LIN {X 0.001,Y -166.682,Z 591.348,A 0.000,B 0.000,C 90.000,E1 242.692} C_DIS
LIN {X -0.008,Y -162.664,Z 591.324,A 0.000,B 0.000,C 90.000,E1 238.329} C_DIS
LIN {X -0.035,Y -161.353,Z 591.314,A 0.000,B 0.000,C 90.000,E1 236.580} C_DIS
LIN {X -0.001,Y -157.347,Z 591.290,A 0.000,B 0.000,C 90.000,E1 232.145} C_DIS
LIN {X 0.028,Y -155.334,Z 591.275,A 0.000,B 0.000,C 90.000,E1 229.461} C_DIS
LIN {X -0.042,Y -151.684,Z 591.250,A 0.000,B 0.000,C 90.000,E1 225.000} C_DIS
LIN {X 0.006,Y -150.547,Z 591.240,A 0.000,B 0.000,C 90.000,E1 223.176} C_DIS
LIN {X 0.039,Y -147.274,Z 591.215,A 0.000,B 0.000,C 90.000,E1 218.624} C_DIS
LIN {X 0.012,Y -145.301,Z 591.194,A 0.000,B 0.000,C 90.000,E1 214.978} C_DIS
LIN {X 0.004,Y -142.395,Z 591.164,A 0.000,B 0.000,C 90.000,E1 209.461} C_DIS
LIN {X -0.014,Y -141.376,Z 591.148,A 0.000,B 0.000,C 90.000,E1 206.693} C_DIS
LIN {X 0.028,Y -139.348,Z 591.112,A 0.000,B 0.000,C 90.000,E1 200.174} C_DIS
LIN {X -0.031,Y -138.784,Z 591.097,A 0.000,B 0.000,C 90.000,E1 197.402} C_DIS
LIN {X 0.028,Y -138.343,Z 591.055,A 0.000,B 0.000,C 90.000,E1 189.905} C_DIS
LIN {X 0.048,Y -139.390,Z 591.008,A 0.000,B 0.000,C 90.000,E1 181.489} C_DIS
LIN {X -0.039,Y -141.288,Z 590.972,A 0.000,B 0.000,C 90.000,E1 175.008} C_DIS
LIN {X 0.061,Y -142.651,Z 590.957,A 0.000,B 0.000,C 90.000,E1 172.186} C_DIS
LIN {X 0.010,Y -144.990,Z 590.931,A 0.000,B 0.000,C 90.000,E1 167.589} C_DIS
LIN {X 0.001,Y -147.617,Z 590.911,A 0.000,B 0.000,C 90.000,E1 163.921} C_DIS
LIN {X 0.079,Y -150.242,Z 590.890,A 0.000,B 0.000,C 90.000,E1 160.242} C_DIS
LIN {X -0.047,Y -153.635,Z 590.870,A 0.000,B 0.000,C 90.000,E1 156.666} C_DIS
LIN {X 0.011,Y -157.051,Z 590.850,A 0.000,B 0.000,C 90.000,E1 153.050} C_DIS
LIN {X 0.009,Y -161.179,Z 590.831,A 0.000,B 0.000,C 90.000,E1 149.488} C_DIS
LIN {X 0.039,Y -163.273,Z 590.821,A 0.000,B 0.000,C 90.000,E1 147.709} C_DIS
LIN {X 0.050,Y -167.715,Z 590.801,A 0.000,B 0.000,C 90.000,E1 144.196} C_DIS
LIN {X -0.037,Y -171.534,Z 590.787,A 0.000,B 0.000,C 90.000,E1 141.618} C_DIS
LIN {X 0.006,Y -176.474,Z 590.768,A 0.000,B 0.000,C 90.000,E1 138.162} C_DIS
LIN {X 0.005,Y -180.771,Z 590.753,A 0.000,B 0.000,C 90.000,E1 135.607} C_DIS
LIN {X -0.008,Y -186.178,Z 590.735,A 0.000,B 0.000,C 90.000,E1 132.243} C_DIS
LIN {X -0.017,Y -191.384,Z 590.719,A 0.000,B 0.000,C 90.000,E1 129.402} C_DIS
LIN {X -0.061,Y -288.933,Z 590.719,A 0.000,B 0.000,C 90.000,E1 129.402} C_DIS
LIN {X -0.121,Y -291.320,Z 590.719,A 0.000,B 0.000,C 90.000,E1 129.358} C_DIS
LIN {X 0.044,Y -295.133,Z 590.717,A 0.000,B 0.000,C 90.000,E1 129.116} C_DIS
LIN {X 0.024,Y -297.460,Z 590.716,A 0.000,B 0.000,C 90.000,E1 128.910} C_DIS
LIN {X 0.053,Y -301.291,Z 590.713,A 0.000,B 0.000,C 90.000,E1 128.382} C_DIS
LIN {X 0.049,Y -302.982,Z 590.711,A 0.000,B 0.000,C 90.000,E1 128.051} C_DIS
LIN {X -0.008,Y -304.309,Z 590.710,A 0.000,B 0.000,C 90.000,E1 127.729} C_DIS
LIN {X 0.022,Y -313.953,Z 590.691,A 0.000,B 0.000,C 90.000,E1 124.452} C_DIS
LIN {X 0.123,Y -323.776,Z 590.675,A 0.000,B 0.000,C 90.000,E1 121.544} C_DIS
LIN {X -0.106,Y -334.914,Z 590.660,A 0.000,B 0.000,C 90.000,E1 118.743} C_DIS
LIN {X 0.095,Y -347.463,Z 590.644,A 0.000,B 0.000,C 90.000,E1 115.924} C_DIS
LIN {X -0.003,Y -359.895,Z 590.631,A 0.000,B 0.000,C 90.000,E1 113.515} C_DIS
LIN {X -0.093,Y -373.621,Z 590.617,A 0.000,B 0.000,C 90.000,E1 111.153} C_DIS
LIN {X -0.121,Y -388.742,Z 590.605,A 0.000,B 0.000,C 90.000,E1 108.833} C_DIS
LIN {X -0.019,Y -405.367,Z 590.592,A 0.000,B 0.000,C 90.000,E1 106.551} C_DIS
LIN {X -0.121,Y -423.616,Z 590.580,A 0.000,B 0.000,C 90.000,E1 104.356} C_DIS
LIN {X -0.201,Y -443.370,Z 590.568,A 0.000,B 0.000,C 90.000,E1 102.243} C_DIS
LIN {X 0.076,Y -463.790,Z 590.557,A 0.000,B 0.000,C 90.000,E1 100.254} C_DIS
LIN {X 0.219,Y -474.052,Z 590.552,A 0.000,B 0.000,C 90.000,E1 99.321} C_DIS
LIN {X -0.232,Y -475.936,Z 590.551,A 0.000,B 0.000,C 90.000,E1 99.151} C_DIS
LIN {X 0.102,Y -477.544,Z 590.549,A 0.000,B 0.000,C 90.000,E1 98.859} C_DIS
LIN {X -0.036,Y -478.750,Z 590.548,A 0.000,B 0.000,C 90.000,E1 98.624} C_DIS
LIN {X 0.110,Y -480.218,Z 590.545,A 0.000,B 0.000,C 90.000,E1 98.106} C_DIS
LIN {X -0.212,Y -480.647,Z 590.542,A 0.000,B 0.000,C 90.000,E1 97.644} C_DIS
LIN {X -0.048,Y -480.105,Z 590.540,A 0.000,B 0.000,C 90.000,E1 97.125} C_DIS
LIN {X 0.119,Y -478.511,Z 590.537,A 0.000,B 0.000,C 90.000,E1 96.606} C_DIS
LIN {X -0.010,Y -477.230,Z 590.535,A 0.000,B 0.000,C 90.000,E1 96.372} C_DIS
LIN {X 0.142,Y -473.633,Z 590.533,A 0.000,B 0.000,C 90.000,E1 95.853} C_DIS
LIN {X 0.030,Y -459.012,Z 590.521,A 0.000,B 0.000,C 90.000,E1 93.841} C_DIS
LIN {X -0.195,Y -447.691,Z 590.511,A 0.000,B 0.000,C 90.000,E1 92.064} C_DIS
LIN {X -0.018,Y -436.085,Z 590.500,A 0.000,B 0.000,C 90.000,E1 89.943} C_DIS
LIN {X -0.110,Y -428.555,Z 590.492,A 0.000,B 0.000,C 90.000,E1 88.625} C_DIS
LIN {X -0.182,Y -419.081,Z 590.483,A 0.000,B 0.000,C 90.000,E1 87.020} C_DIS
LIN {X -0.058,Y -403.319,Z 590.468,A 0.000,B 0.000,C 90.000,E1 84.261} C_DIS
LIN {X 0.032,Y -389.890,Z 590.454,A 0.000,B 0.000,C 90.000,E1 81.724} C_DIS
LIN {X -0.088,Y -378.203,Z 590.441,A 0.000,B 0.000,C 90.000,E1 79.454} C_DIS
LIN {X -0.056,Y -365.412,Z 590.427,A 0.000,B 0.000,C 90.000,E1 76.825} C_DIS
LIN {X -0.079,Y -351.916,Z 590.410,A 0.000,B 0.000,C 90.000,E1 73.850} C_DIS
LIN {X 0.043,Y -339.732,Z 590.393,A 0.000,B 0.000,C 90.000,E1 70.786} C_DIS
LIN {X 0.158,Y -329.793,Z 590.378,A 0.000,B 0.000,C 90.000,E1 67.975} C_DIS
LIN {X 0.040,Y -319.831,Z 590.360,A 0.000,B 0.000,C 90.000,E1 64.845} C_DIS
LIN {X 0.058,Y -312.250,Z 590.346,A 0.000,B 0.000,C 90.000,E1 62.281} C_DIS
LIN {X 0.176,Y -304.903,Z 590.332,A 0.000,B 0.000,C 90.000,E1 59.665} C_DIS
LIN {X 0.152,Y -297.769,Z 590.317,A 0.000,B 0.000,C 90.000,E1 57.041} C_DIS
LIN {X -0.058,Y -289.305,Z 590.299,A 0.000,B 0.000,C 90.000,E1 53.749} C_DIS
LIN {X 0.077,Y -284.390,Z 590.287,A 0.000,B 0.000,C 90.000,E1 51.698} C_DIS
LIN {X 0.022,Y -279.299,Z 590.276,A 0.000,B 0.000,C 90.000,E1 49.666} C_DIS
LIN {X -0.123,Y -275.670,Z 590.268,A 0.000,B 0.000,C 90.000,E1 48.324} C_DIS
LIN {X 0.052,Y -271.817,Z 590.261,A 0.000,B 0.000,C 90.000,E1 46.905} C_DIS
LIN {X -0.010,Y -267.604,Z 590.253,A 0.000,B 0.000,C 90.000,E1 45.526} C_DIS
LIN {X -0.022,Y -260.833,Z 590.241,A 0.000,B 0.000,C 90.000,E1 43.419} C_DIS
LIN {X 0.032,Y -252.799,Z 590.227,A 0.000,B 0.000,C 90.000,E1 40.906} C_DIS
LIN {X -0.030,Y -242.966,Z 590.209,A 0.000,B 0.000,C 90.000,E1 37.649} C_DIS
LIN {X -0.027,Y -235.024,Z 590.193,A 0.000,B 0.000,C 90.000,E1 34.692} C_DIS
LIN {X 0.037,Y -227.788,Z 590.176,A 0.000,B 0.000,C 90.000,E1 31.671} C_DIS
LIN {X 0.065,Y -221.233,Z 590.159,A 0.000,B 0.000,C 90.000,E1 28.615} C_DIS
LIN {X 0.005,Y -215.441,Z 590.142,A 0.000,B 0.000,C 90.000,E1 25.540} C_DIS
LIN {X 0.018,Y -210.399,Z 590.125,A 0.000,B 0.000,C 90.000,E1 22.408} C_DIS
LIN {X -0.052,Y -205.263,Z 590.103,A 0.000,B 0.000,C 90.000,E1 18.471} C_DIS
LIN {X -0.080,Y -201.272,Z 590.080,A 0.000,B 0.000,C 90.000,E1 14.481} C_DIS
LIN {X 0.013,Y -197.803,Z 590.053,A 0.000,B 0.000,C 90.000,E1 9.613} C_DIS
LIN {X 0.016,Y -195.578,Z 590.013,A 0.000,B 0.000,C 90.000,E1 2.293} C_DIS
LIN {X 0.101,Y -197.278,Z 589.966,A 0.000,B 0.000,C 90.000,E1 353.799} C_DIS
LIN {X -0.074,Y -200.204,Z 589.939,A 0.000,B 0.000,C 90.000,E1 348.982} C_DIS
LIN {X -0.099,Y -204.480,Z 589.912,A 0.000,B 0.000,C 90.000,E1 344.157} C_DIS
LIN {X 0.015,Y -208.872,Z 589.890,A 0.000,B 0.000,C 90.000,E1 340.134} C_DIS
LIN {X 0.037,Y -214.099,Z 589.868,A 0.000,B 0.000,C 90.000,E1 336.177} C_DIS
LIN {X -0.003,Y -220.025,Z 589.846,A 0.000,B 0.000,C 90.000,E1 332.281} C_DIS
LIN {X 0.066,Y -226.572,Z 589.825,A 0.000,B 0.000,C 90.000,E1 328.408} C_DIS
LIN {X -0.044,Y -232.201,Z 589.808,A 0.000,B 0.000,C 90.000,E1 325.388} C_DIS
LIN {X 0.004,Y -239.520,Z 589.787,A 0.000,B 0.000,C 90.000,E1 321.618} C_DIS
LIN {X -0.014,Y -247.551,Z 589.766,A 0.000,B 0.000,C 90.000,E1 317.919} C_DIS
LIN {X 0.014,Y -256.490,Z 589.746,A 0.000,B 0.000,C 90.000,E1 314.271} C_DIS
LIN {X -0.004,Y -266.682,Z 589.726,A 0.000,B 0.000,C 90.000,E1 310.701} C_DIS
LIN {X 0.028,Y -276.166,Z 589.711,A 0.000,B 0.000,C 90.000,E1 307.890} C_DIS
LIN {X -0.108,Y -289.433,Z 589.691,A 0.000,B 0.000,C 90.000,E1 304.485} C_DIS
LIN {X -0.071,Y -304.313,Z 589.673,A 0.000,B 0.000,C 90.000,E1 301.131} C_DIS
LIN {X 0.103,Y -317.089,Z 589.658,A 0.000,B 0.000,C 90.000,E1 298.487} C_DIS
LIN {X -0.070,Y -333.996,Z 589.641,A 0.000,B 0.000,C 90.000,E1 295.335} C_DIS
LIN {X 0.135,Y -348.856,Z 589.627,A 0.000,B 0.000,C 90.000,E1 292.823} C_DIS
LIN {X -0.003,Y -365.106,Z 589.613,A 0.000,B 0.000,C 90.000,E1 290.429} C_DIS
LIN {X 0.155,Y -385.211,Z 589.599,A 0.000,B 0.000,C 90.000,E1 287.764} C_DIS
LIN {X -0.042,Y -399.377,Z 589.589,A 0.000,B 0.000,C 90.000,E1 286.079} C_DIS
LIN {X -0.112,Y -413.409,Z 589.580,A 0.000,B 0.000,C 90.000,E1 284.411} C_DIS
LIN {X -0.131,Y -427.361,Z 589.571,A 0.000,B 0.000,C 90.000,E1 282.771} C_DIS
LIN {X 0.145,Y -436.179,Z 589.565,A 0.000,B 0.000,C 90.000,E1 281.658} C_DIS
LIN {X 0.101,Y -444.479,Z 589.559,A 0.000,B 0.000,C 90.000,E1 280.602} C_DIS
LIN {X 0.070,Y -452.385,Z 589.553,A 0.000,B 0.000,C 90.000,E1 279.557} C_DIS
LIN {X -0.139,Y -457.960,Z 589.549,A 0.000,B 0.000,C 90.000,E1 278.803} C_DIS
LIN {X -0.015,Y -464.839,Z 589.543,A 0.000,B 0.000,C 90.000,E1 277.757} C_DIS
LIN {X 0.129,Y -471.173,Z 589.537,A 0.000,B 0.000,C 90.000,E1 276.720} C_DIS
LIN {X 0.081,Y -475.463,Z 589.533,A 0.000,B 0.000,C 90.000,E1 275.967} C_DIS
LIN {X 0.013,Y -479.078,Z 589.529,A 0.000,B 0.000,C 90.000,E1 275.220} C_DIS
LIN {X 0.162,Y -481.108,Z 589.526,A 0.000,B 0.000,C 90.000,E1 274.702} C_DIS
LIN {X -0.200,Y -482.801,Z 589.523,A 0.000,B 0.000,C 90.000,E1 274.245} C_DIS
LIN {X -0.034,Y -484.173,Z 589.521,A 0.000,B 0.000,C 90.000,E1 273.726} C_DIS
LIN {X 0.112,Y -485.263,Z 589.518,A 0.000,B 0.000,C 90.000,E1 273.212} C_DIS
LIN {X -0.192,Y -486.019,Z 589.515,A 0.000,B 0.000,C 90.000,E1 272.751} C_DIS
LIN {X -0.028,Y -486.481,Z 589.512,A 0.000,B 0.000,C 90.000,E1 272.236} C_DIS
LIN {X 0.158,Y -486.570,Z 589.510,A 0.000,B 0.000,C 90.000,E1 271.718} C_DIS
LIN {X -0.157,Y -486.200,Z 589.507,A 0.000,B 0.000,C 90.000,E1 271.260} C_DIS
LIN {X 0.017,Y -485.368,Z 589.504,A 0.000,B 0.000,C 90.000,E1 270.745} C_DIS
LIN {X 0.189,Y -484.045,Z 589.501,A 0.000,B 0.000,C 90.000,E1 270.229} C_DIS
LIN {X -0.127,Y -482.086,Z 589.499,A 0.000,B 0.000,C 90.000,E1 269.771} C_DIS
LIN {X 0.032,Y -479.359,Z 589.496,A 0.000,B 0.000,C 90.000,E1 269.255} C_DIS
LIN {X -0.137,Y -477.707,Z 589.495,A 0.000,B 0.000,C 90.000,E1 269.026} C_DIS
LIN {X -0.008,Y -473.588,Z 589.492,A 0.000,B 0.000,C 90.000,E1 268.511} C_DIS
LIN {X -0.185,Y -471.206,Z 589.490,A 0.000,B 0.000,C 90.000,E1 268.282} C_DIS
LIN {X -0.073,Y -465.267,Z 589.488,A 0.000,B 0.000,C 90.000,E1 267.764} C_DIS
LIN {X 0.141,Y -458.882,Z 589.485,A 0.000,B 0.000,C 90.000,E1 267.306} C_DIS
LIN {X -0.018,Y -451.775,Z 589.483,A 0.000,B 0.000,C 90.000,E1 266.963} C_DIS
LIN {X 0.003,Y -444.612,Z 589.482,A 0.000,B 0.000,C 90.000,E1 266.674} C_DIS
LIN {X -0.015,Y -436.746,Z 589.480,A 0.000,B 0.000,C 90.000,E1 266.445} C_DIS
LIN {X -0.018,Y -428.223,Z 589.479,A 0.000,B 0.000,C 90.000,E1 266.274} C_DIS
LIN {X -0.045,Y -418.357,Z 589.479,A 0.000,B 0.000,C 90.000,E1 266.159} C_DIS
LIN {X -0.061,Y -408.534,Z 589.478,A 0.000,B 0.000,C 90.000,E1 266.102} C_DIS
LIN {X -0.058,Y -180.923,Z 589.478,A 0.000,B 0.000,C 90.000,E1 266.102} C_DIS
LIN {X -0.013,Y -180.875,Z 589.473,A 0.000,B 0.000,C 90.000,E1 265.065} C_DIS
LIN {X 0.069,Y -178.940,Z 589.443,A 0.000,B 0.000,C 90.000,E1 259.803} C_DIS
LIN {X -0.063,Y -175.990,Z 589.415,A 0.000,B 0.000,C 90.000,E1 254.755} C_DIS
LIN {X 0.052,Y -175.491,Z 589.410,A 0.000,B 0.000,C 90.000,E1 253.866} C_DIS
LIN {X -0.054,Y -172.235,Z 589.387,A 0.000,B 0.000,C 90.000,E1 249.625} C_DIS
LIN {X -0.075,Y -171.712,Z 589.382,A 0.000,B 0.000,C 90.000,E1 248.773} C_DIS
LIN {X 0.010,Y -167.307,Z 589.353,A 0.000,B 0.000,C 90.000,E1 243.563} C_DIS
LIN {X 0.016,Y -166.687,Z 589.348,A 0.000,B 0.000,C 90.000,E1 242.692} C_DIS
LIN {X 0.006,Y -162.668,Z 589.324,A 0.000,B 0.000,C 90.000,E1 238.329} C_DIS
LIN {X -0.020,Y -161.358,Z 589.314,A 0.000,B 0.000,C 90.000,E1 236.580} C_DIS
LIN {X 0.014,Y -157.351,Z 589.290,A 0.000,B 0.000,C 90.000,E1 232.145} C_DIS
LIN {X 0.043,Y -155.339,Z 589.275,A 0.000,B 0.000,C 90.000,E1 229.461} C_DIS
LIN {X -0.028,Y -151.688,Z 589.250,A 0.000,B 0.000,C 90.000,E1 225.000} C_DIS
LIN {X 0.021,Y -150.551,Z 589.240,A 0.000,B 0.000,C 90.000,E1 223.176} C_DIS
LIN {X 0.053,Y -147.277,Z 589.215,A 0.000,B 0.000,C 90.000,E1 218.624} C_DIS
LIN {X 0.026,Y -145.305,Z 589.194,A 0.000,B 0.000,C 90.000,E1 214.978} C_DIS
LIN {X 0.017,Y -142.398,Z 589.164,A 0.000,B 0.000,C 90.000,E1 209.461} C_DIS
LIN {X 0.000,Y -141.378,Z 589.148,A 0.000,B 0.000,C 90.000,E1 206.693} C_DIS
LIN {X 0.041,Y -139.348,Z 589.112,A 0.000,B 0.000,C 90.000,E1 200.174} C_DIS
LIN {X -0.018,Y -138.785,Z 589.097,A 0.000,B 0.000,C 90.000,E1 197.402} C_DIS
LIN {X 0.041,Y -138.344,Z 589.055,A 0.000,B 0.000,C 90.000,E1 189.905} C_DIS
LIN {X 0.062,Y -139.389,Z 589.008,A 0.000,B 0.000,C 90.000,E1 181.489} C_DIS
LIN {X -0.025,Y -141.285,Z 588.972,A 0.000,B 0.000,C 90.000,E1 175.008} C_DIS
LIN {X -0.067,Y -142.649,Z 588.957,A 0.000,B 0.000,C 90.000,E1 172.243} C_DIS
LIN {X 0.025,Y -144.986,Z 588.931,A 0.000,B 0.000,C 90.000,E1 167.589} C_DIS
LIN {X 0.014,Y -147.614,Z 588.911,A 0.000,B 0.000,C 90.000,E1 163.921} C_DIS
LIN {X -0.048,Y -150.237,Z 588.890,A 0.000,B 0.000,C 90.000,E1 160.296} C_DIS
LIN {X -0.032,Y -153.630,Z 588.870,A 0.000,B 0.000,C 90.000,E1 156.666} C_DIS
LIN {X 0.026,Y -157.046,Z 588.850,A 0.000,B 0.000,C 90.000,E1 153.050} C_DIS
LIN {X 0.025,Y -161.172,Z 588.831,A 0.000,B 0.000,C 90.000,E1 149.488} C_DIS
LIN {X -0.033,Y -163.267,Z 588.821,A 0.000,B 0.000,C 90.000,E1 147.740} C_DIS
LIN {X 0.066,Y -167.707,Z 588.801,A 0.000,B 0.000,C 90.000,E1 144.196} C_DIS
LIN {X -0.021,Y -171.527,Z 588.787,A 0.000,B 0.000,C 90.000,E1 141.618} C_DIS
LIN {X 0.022,Y -176.467,Z 588.768,A 0.000,B 0.000,C 90.000,E1 138.162} C_DIS
LIN {X -0.109,Y -180.763,Z 588.753,A 0.000,B 0.000,C 90.000,E1 135.648} C_DIS
LIN {X 0.010,Y -186.169,Z 588.735,A 0.000,B 0.000,C 90.000,E1 132.243} C_DIS
LIN {X -0.002,Y -191.377,Z 588.719,A 0.000,B 0.000,C 90.000,E1 129.402} C_DIS
LIN {X -0.048,Y -191.400,Z 588.719,A 0.000,B 0.000,C 90.000,E1 129.402} C_DIS
LIN {X 0.115,Y -288.729,Z 588.719,A 0.000,B 0.000,C 90.000,E1 129.358} C_DIS
LIN {X -0.096,Y -290.833,Z 588.719,A 0.000,B 0.000,C 90.000,E1 129.358} C_DIS
LIN {X 0.069,Y -294.924,Z 588.717,A 0.000,B 0.000,C 90.000,E1 129.116} C_DIS
LIN {X 0.050,Y -297.311,Z 588.716,A 0.000,B 0.000,C 90.000,E1 128.910} C_DIS
LIN {X 0.138,Y -301.139,Z 588.713,A 0.000,B 0.000,C 90.000,E1 128.382} C_DIS
LIN {X -0.104,Y -302.866,Z 588.712,A 0.000,B 0.000,C 90.000,E1 128.096} C_DIS
LIN {X 0.077,Y -304.220,Z 588.710,A 0.000,B 0.000,C 90.000,E1 127.729} C_DIS
LIN {X -0.161,Y -309.912,Z 588.699,A 0.000,B 0.000,C 90.000,E1 125.804} C_DIS
LIN {X -0.039,Y -320.286,Z 588.681,A 0.000,B 0.000,C 90.000,E1 122.546} C_DIS
LIN {X 0.082,Y -330.967,Z 588.665,A 0.000,B 0.000,C 90.000,E1 119.667} C_DIS
LIN {X 0.021,Y -343.028,Z 588.649,A 0.000,B 0.000,C 90.000,E1 116.873} C_DIS
LIN {X -0.006,Y -356.570,Z 588.634,A 0.000,B 0.000,C 90.000,E1 114.131} C_DIS
LIN {X 0.160,Y -369.957,Z 588.621,A 0.000,B 0.000,C 90.000,E1 111.716} C_DIS
LIN {X 0.061,Y -384.711,Z 588.608,A 0.000,B 0.000,C 90.000,E1 109.396} C_DIS
LIN {X 0.200,Y -400.939,Z 588.595,A 0.000,B 0.000,C 90.000,E1 107.094} C_DIS
LIN {X 0.003,Y -418.761,Z 588.583,A 0.000,B 0.000,C 90.000,E1 104.898} C_DIS
LIN {X -0.206,Y -438.211,Z 588.571,A 0.000,B 0.000,C 90.000,E1 102.771} C_DIS
LIN {X 0.170,Y -458.490,Z 588.560,A 0.000,B 0.000,C 90.000,E1 100.725} C_DIS
LIN {X -0.166,Y -473.947,Z 588.552,A 0.000,B 0.000,C 90.000,E1 99.378} C_DIS
LIN {X -0.150,Y -475.883,Z 588.551,A 0.000,B 0.000,C 90.000,E1 99.151} C_DIS
LIN {X 0.184,Y -477.532,Z 588.549,A 0.000,B 0.000,C 90.000,E1 98.859} C_DIS
LIN {X 0.047,Y -478.768,Z 588.548,A 0.000,B 0.000,C 90.000,E1 98.624} C_DIS
LIN {X 0.191,Y -480.289,Z 588.545,A 0.000,B 0.000,C 90.000,E1 98.106} C_DIS
LIN {X -0.130,Y -480.762,Z 588.542,A 0.000,B 0.000,C 90.000,E1 97.644} C_DIS
LIN {X 0.034,Y -480.265,Z 588.540,A 0.000,B 0.000,C 90.000,E1 97.125} C_DIS
LIN {X 0.201,Y -478.721,Z 588.537,A 0.000,B 0.000,C 90.000,E1 96.606} C_DIS
LIN {X 0.072,Y -477.474,Z 588.535,A 0.000,B 0.000,C 90.000,E1 96.372} C_DIS
LIN {X 0.225,Y -473.905,Z 588.533,A 0.000,B 0.000,C 90.000,E1 95.853} C_DIS
LIN {X 0.116,Y -459.250,Z 588.521,A 0.000,B 0.000,C 90.000,E1 93.841} C_DIS
LIN {X 0.132,Y -449.400,Z 588.513,A 0.000,B 0.000,C 90.000,E1 92.293} C_DIS
LIN {X -0.199,Y -434.797,Z 588.498,A 0.000,B 0.000,C 90.000,E1 89.714} C_DIS
LIN {X 0.124,Y -427.168,Z 588.491,A 0.000,B 0.000,C 90.000,E1 88.339} C_DIS
LIN {X 0.144,Y -416.037,Z 588.480,A 0.000,B 0.000,C 90.000,E1 86.445} C_DIS
LIN {X -0.140,Y -398.934,Z 588.464,A 0.000,B 0.000,C 90.000,E1 83.451} C_DIS
LIN {X -0.152,Y -387.064,Z 588.451,A 0.000,B 0.000,C 90.000,E1 81.197} C_DIS
LIN {X 0.055,Y -373.987,Z 588.437,A 0.000,B 0.000,C 90.000,E1 78.578} C_DIS
LIN {X 0.054,Y -361.295,Z 588.422,A 0.000,B 0.000,C 90.000,E1 75.936} C_DIS
LIN {X -0.089,Y -348.159,Z 588.405,A 0.000,B 0.000,C 90.000,E1 72.960} C_DIS
LIN {X 0.003,Y -334.154,Z 588.385,A 0.000,B 0.000,C 90.000,E1 69.263} C_DIS
LIN {X 0.097,Y -321.865,Z 588.364,A 0.000,B 0.000,C 90.000,E1 65.485} C_DIS
LIN {X 0.018,Y -314.223,Z 588.350,A 0.000,B 0.000,C 90.000,E1 62.948} C_DIS
LIN {X -0.089,Y -306.840,Z 588.335,A 0.000,B 0.000,C 90.000,E1 60.383} C_DIS
LIN {X 0.042,Y -299.628,Z 588.321,A 0.000,B 0.000,C 90.000,E1 57.740} C_DIS
LIN {X 0.121,Y -291.023,Z 588.302,A 0.000,B 0.000,C 90.000,E1 54.402} C_DIS
LIN {X 0.059,Y -286.111,Z 588.291,A 0.000,B 0.000,C 90.000,E1 52.396} C_DIS
LIN {X 0.079,Y -281.088,Z 588.280,A 0.000,B 0.000,C 90.000,E1 50.356} C_DIS
LIN {X -0.046,Y -277.588,Z 588.272,A 0.000,B 0.000,C 90.000,E1 49.013} C_DIS
LIN {X -0.045,Y -271.877,Z 588.261,A 0.000,B 0.000,C 90.000,E1 46.944} C_DIS
LIN {X 0.145,Y -266.552,Z 588.251,A 0.000,B 0.000,C 90.000,E1 45.162} C_DIS
LIN {X 0.141,Y -258.564,Z 588.237,A 0.000,B 0.000,C 90.000,E1 42.690} C_DIS
LIN {X 0.006,Y -248.295,Z 588.219,A 0.000,B 0.000,C 90.000,E1 39.483} C_DIS
LIN {X 0.069,Y -238.916,Z 588.201,A 0.000,B 0.000,C 90.000,E1 36.171} C_DIS
LIN {X -0.028,Y -231.325,Z 588.185,A 0.000,B 0.000,C 90.000,E1 33.214} C_DIS
LIN {X -0.108,Y -224.424,Z 588.168,A 0.000,B 0.000,C 90.000,E1 30.207} C_DIS
LIN {X -0.075,Y -218.224,Z 588.151,A 0.000,B 0.000,C 90.000,E1 27.129} C_DIS
LIN {X -0.014,Y -212.811,Z 588.133,A 0.000,B 0.000,C 90.000,E1 24.003} C_DIS
LIN {X -0.039,Y -208.167,Z 588.116,A 0.000,B 0.000,C 90.000,E1 20.865} C_DIS
LIN {X 0.075,Y -203.500,Z 588.094,A 0.000,B 0.000,C 90.000,E1 16.858} C_DIS
LIN {X -0.011,Y -199.334,Z 588.067,A 0.000,B 0.000,C 90.000,E1 12.063} C_DIS
LIN {X 0.051,Y -196.338,Z 588.035,A 0.000,B 0.000,C 90.000,E1 6.372} C_DIS
LIN {X 0.068,Y -197.666,Z 587.961,A 0.000,B 0.000,C 90.000,E1 352.996} C_DIS
LIN {X -0.072,Y -200.861,Z 587.934,A 0.000,B 0.000,C 90.000,E1 348.173} C_DIS
LIN {X -0.098,Y -204.508,Z 587.912,A 0.000,B 0.000,C 90.000,E1 344.157} C_DIS
LIN {X 0.016,Y -208.889,Z 587.890,A 0.000,B 0.000,C 90.000,E1 340.134} C_DIS
LIN {X 0.038,Y -214.124,Z 587.868,A 0.000,B 0.000,C 90.000,E1 336.177} C_DIS
LIN {X 0.000,Y -220.047,Z 587.846,A 0.000,B 0.000,C 90.000,E1 332.281} C_DIS
LIN {X 0.070,Y -226.564,Z 587.825,A 0.000,B 0.000,C 90.000,E1 328.408} C_DIS
LIN {X -0.041,Y -232.172,Z 587.808,A 0.000,B 0.000,C 90.000,E1 325.388} C_DIS
LIN {X 0.006,Y -239.507,Z 587.787,A 0.000,B 0.000,C 90.000,E1 321.618} C_DIS
LIN {X -0.012,Y -247.539,Z 587.766,A 0.000,B 0.000,C 90.000,E1 317.919} C_DIS
LIN {X 0.016,Y -256.456,Z 587.746,A 0.000,B 0.000,C 90.000,E1 314.271} C_DIS
LIN {X -0.003,Y -266.631,Z 587.726,A 0.000,B 0.000,C 90.000,E1 310.701} C_DIS
LIN {X 0.028,Y -276.135,Z 587.711,A 0.000,B 0.000,C 90.000,E1 307.890} C_DIS
LIN {X -0.109,Y -289.396,Z 587.691,A 0.000,B 0.000,C 90.000,E1 304.485} C_DIS
LIN {X -0.074,Y -304.254,Z 587.673,A 0.000,B 0.000,C 90.000,E1 301.131} C_DIS
LIN {X 0.098,Y -316.989,Z 587.658,A 0.000,B 0.000,C 90.000,E1 298.487} C_DIS
LIN {X -0.038,Y -332.113,Z 587.642,A 0.000,B 0.000,C 90.000,E1 295.643} C_DIS
LIN {X -0.022,Y -346.809,Z 587.629,A 0.000,B 0.000,C 90.000,E1 293.153} C_DIS
LIN {X -0.017,Y -365.059,Z 587.613,A 0.000,B 0.000,C 90.000,E1 290.429} C_DIS
LIN {X 0.138,Y -385.186,Z 587.599,A 0.000,B 0.000,C 90.000,E1 287.764} C_DIS
LIN {X -0.060,Y -399.381,Z 587.589,A 0.000,B 0.000,C 90.000,E1 286.079} C_DIS
LIN {X -0.130,Y -413.427,Z 587.580,A 0.000,B 0.000,C 90.000,E1 284.411} C_DIS
LIN {X 0.108,Y -425.114,Z 587.572,A 0.000,B 0.000,C 90.000,E1 283.008} C_DIS
LIN {X -0.063,Y -434.074,Z 587.566,A 0.000,B 0.000,C 90.000,E1 281.951} C_DIS
LIN {X -0.134,Y -442.496,Z 587.560,A 0.000,B 0.000,C 90.000,E1 280.894} C_DIS
LIN {X -0.192,Y -450.502,Z 587.555,A 0.000,B 0.000,C 90.000,E1 279.849} C_DIS
LIN {X 0.109,Y -456.221,Z 587.550,A 0.000,B 0.000,C 90.000,E1 279.029} C_DIS
LIN {X 0.147,Y -463.228,Z 587.544,A 0.000,B 0.000,C 90.000,E1 277.992} C_DIS
LIN {X -0.132,Y -469.696,Z 587.539,A 0.000,B 0.000,C 90.000,E1 277.004} C_DIS
LIN {X 0.065,Y -475.471,Z 587.533,A 0.000,B 0.000,C 90.000,E1 275.967} C_DIS
LIN {X -0.002,Y -479.099,Z 587.529,A 0.000,B 0.000,C 90.000,E1 275.220} C_DIS
LIN {X 0.147,Y -481.116,Z 587.526,A 0.000,B 0.000,C 90.000,E1 274.702} C_DIS
LIN {X -0.216,Y -482.801,Z 587.523,A 0.000,B 0.000,C 90.000,E1 274.245} C_DIS
LIN {X -0.049,Y -484.212,Z 587.521,A 0.000,B 0.000,C 90.000,E1 273.726} C_DIS
LIN {X 0.097,Y -485.302,Z 587.518,A 0.000,B 0.000,C 90.000,E1 273.212} C_DIS
LIN {X -0.207,Y -486.096,Z 587.515,A 0.000,B 0.000,C 90.000,E1 272.751} C_DIS
LIN {X -0.043,Y -486.575,Z 587.512,A 0.000,B 0.000,C 90.000,E1 272.236} C_DIS
LIN {X 0.143,Y -486.642,Z 587.510,A 0.000,B 0.000,C 90.000,E1 271.718} C_DIS
LIN {X -0.171,Y -486.248,Z 587.507,A 0.000,B 0.000,C 90.000,E1 271.260} C_DIS
LIN {X 0.004,Y -485.425,Z 587.504,A 0.000,B 0.000,C 90.000,E1 270.745} C_DIS
LIN {X 0.176,Y -484.025,Z 587.501,A 0.000,B 0.000,C 90.000,E1 270.229} C_DIS
LIN {X -0.140,Y -482.076,Z 587.499,A 0.000,B 0.000,C 90.000,E1 269.771} C_DIS
LIN {X 0.019,Y -479.361,Z 587.496,A 0.000,B 0.000,C 90.000,E1 269.255} C_DIS
LIN {X 0.157,Y -475.810,Z 587.493,A 0.000,B 0.000,C 90.000,E1 268.740} C_DIS
LIN {X -0.198,Y -471.170,Z 587.490,A 0.000,B 0.000,C 90.000,E1 268.282} C_DIS
LIN {X -0.087,Y -465.256,Z 587.488,A 0.000,B 0.000,C 90.000,E1 267.764} C_DIS
LIN {X 0.019,Y -462.236,Z 587.486,A 0.000,B 0.000,C 90.000,E1 267.535} C_DIS
LIN {X 0.077,Y -455.516,Z 587.484,A 0.000,B 0.000,C 90.000,E1 267.135} C_DIS
LIN {X -0.191,Y -448.463,Z 587.482,A 0.000,B 0.000,C 90.000,E1 266.846} C_DIS
LIN {X 0.003,Y -440.953,Z 587.481,A 0.000,B 0.000,C 90.000,E1 266.560} C_DIS
LIN {X 0.209,Y -432.968,Z 587.480,A 0.000,B 0.000,C 90.000,E1 266.331} C_DIS
LIN {X -0.028,Y -424.153,Z 587.479,A 0.000,B 0.000,C 90.000,E1 266.216} C_DIS
LIN {X 0.081,Y -413.506,Z 587.478,A 0.000,B 0.000,C 90.000,E1 266.102} C_DIS
LIN {X -0.063,Y -408.887,Z 587.478,A 0.000,B 0.000,C 90.000,E1 266.102} C_DIS
LIN {X -0.059,Y -180.924,Z 587.478,A 0.000,B 0.000,C 90.000,E1 266.102} C_DIS
LIN {X -0.014,Y -180.875,Z 587.473,A 0.000,B 0.000,C 90.000,E1 265.065} C_DIS
LIN {X 0.068,Y -178.939,Z 587.443,A 0.000,B 0.000,C 90.000,E1 259.803} C_DIS
LIN {X -0.064,Y -175.990,Z 587.415,A 0.000,B 0.000,C 90.000,E1 254.755} C_DIS
LIN {X 0.050,Y -175.490,Z 587.410,A 0.000,B 0.000,C 90.000,E1 253.866} C_DIS
LIN {X -0.055,Y -172.234,Z 587.387,A 0.000,B 0.000,C 90.000,E1 249.625} C_DIS
LIN {X -0.076,Y -171.711,Z 587.382,A 0.000,B 0.000,C 90.000,E1 248.773} C_DIS
LIN {X 0.009,Y -167.306,Z 587.353,A 0.000,B 0.000,C 90.000,E1 243.563} C_DIS
LIN {X 0.014,Y -166.686,Z 587.348,A 0.000,B 0.000,C 90.000,E1 242.692} C_DIS
LIN {X 0.005,Y -162.668,Z 587.324,A 0.000,B 0.000,C 90.000,E1 238.329} C_DIS
LIN {X -0.021,Y -161.357,Z 587.314,A 0.000,B 0.000,C 90.000,E1 236.580} C_DIS
LIN {X 0.012,Y -157.351,Z 587.290,A 0.000,B 0.000,C 90.000,E1 232.145} C_DIS
LIN {X 0.041,Y -155.339,Z 587.275,A 0.000,B 0.000,C 90.000,E1 229.461} C_DIS
LIN {X -0.029,Y -151.688,Z 587.250,A 0.000,B 0.000,C 90.000,E1 225.000} C_DIS
LIN {X 0.019,Y -150.551,Z 587.240,A 0.000,B 0.000,C 90.000,E1 223.176} C_DIS
LIN {X 0.051,Y -147.276,Z 587.215,A 0.000,B 0.000,C 90.000,E1 218.624} C_DIS
LIN {X 0.024,Y -145.305,Z 587.194,A 0.000,B 0.000,C 90.000,E1 214.978} C_DIS
LIN {X 0.016,Y -142.397,Z 587.164,A 0.000,B 0.000,C 90.000,E1 209.461} C_DIS
LIN {X -0.001,Y -141.378,Z 587.148,A 0.000,B 0.000,C 90.000,E1 206.693} C_DIS
LIN {X 0.039,Y -139.348,Z 587.112,A 0.000,B 0.000,C 90.000,E1 200.174} C_DIS
LIN {X -0.018,Y -138.785,Z 587.097,A 0.000,B 0.000,C 90.000,E1 197.402} C_DIS
LIN {X 0.040,Y -138.344,Z 587.055,A 0.000,B 0.000,C 90.000,E1 189.905} C_DIS
LIN {X 0.060,Y -139.389,Z 587.008,A 0.000,B 0.000,C 90.000,E1 181.489} C_DIS
LIN {X -0.027,Y -141.285,Z 586.972,A 0.000,B 0.000,C 90.000,E1 175.008} C_DIS
LIN {X -0.069,Y -142.650,Z 586.957,A 0.000,B 0.000,C 90.000,E1 172.243} C_DIS
LIN {X 0.023,Y -144.986,Z 586.931,A 0.000,B 0.000,C 90.000,E1 167.589} C_DIS
LIN {X 0.013,Y -147.614,Z 586.911,A 0.000,B 0.000,C 90.000,E1 163.921} C_DIS
LIN {X -0.050,Y -150.238,Z 586.890,A 0.000,B 0.000,C 90.000,E1 160.296} C_DIS
LIN {X -0.034,Y -153.631,Z 586.870,A 0.000,B 0.000,C 90.000,E1 156.666} C_DIS
LIN {X 0.024,Y -157.046,Z 586.850,A 0.000,B 0.000,C 90.000,E1 153.050} C_DIS
LIN {X 0.023,Y -161.173,Z 586.831,A 0.000,B 0.000,C 90.000,E1 149.488} C_DIS
LIN {X -0.034,Y -163.268,Z 586.821,A 0.000,B 0.000,C 90.000,E1 147.740} C_DIS
LIN {X 0.064,Y -167.709,Z 586.801,A 0.000,B 0.000,C 90.000,E1 144.196} C_DIS
LIN {X -0.023,Y -171.528,Z 586.787,A 0.000,B 0.000,C 90.000,E1 141.618} C_DIS
LIN {X 0.020,Y -176.467,Z 586.768,A 0.000,B 0.000,C 90.000,E1 138.162} C_DIS
LIN {X -0.110,Y -180.764,Z 586.753,A 0.000,B 0.000,C 90.000,E1 135.648} C_DIS
LIN {X 0.008,Y -186.170,Z 586.735,A 0.000,B 0.000,C 90.000,E1 132.243} C_DIS
LIN {X -0.004,Y -191.378,Z 586.719,A 0.000,B 0.000,C 90.000,E1 129.402} C_DIS
LIN {X 0.050,Y -191.424,Z 586.719,A 0.000,B 0.000,C 90.000,E1 129.358} C_DIS
LIN {X 0.031,Y -288.925,Z 586.719,A 0.000,B 0.000,C 90.000,E1 129.358} C_DIS
LIN {X -0.101,Y -290.352,Z 586.719,A 0.000,B 0.000,C 90.000,E1 129.358} C_DIS
LIN {X 0.065,Y -294.747,Z 586.717,A 0.000,B 0.000,C 90.000,E1 129.116} C_DIS
LIN {X 0.048,Y -297.190,Z 586.716,A 0.000,B 0.000,C 90.000,E1 128.910} C_DIS
LIN {X 0.001,Y -301.013,Z 586.713,A 0.000,B 0.000,C 90.000,E1 128.418} C_DIS
LIN {X -0.055,Y -302.774,Z 586.712,A 0.000,B 0.000,C 90.000,E1 128.096} C_DIS
LIN {X 0.127,Y -304.153,Z 586.710,A 0.000,B 0.000,C 90.000,E1 127.729} C_DIS
LIN {X 0.079,Y -307.968,Z 586.702,A 0.000,B 0.000,C 90.000,E1 126.423} C_DIS
LIN {X 0.134,Y -318.039,Z 586.684,A 0.000,B 0.000,C 90.000,E1 123.166} C_DIS
LIN {X -0.084,Y -328.422,Z 586.668,A 0.000,B 0.000,C 90.000,E1 120.335} C_DIS
LIN {X -0.061,Y -340.164,Z 586.653,A 0.000,B 0.000,C 90.000,E1 117.513} C_DIS
LIN {X -0.173,Y -353.362,Z 586.637,A 0.000,B 0.000,C 90.000,E1 114.771} C_DIS
LIN {X 0.051,Y -366.418,Z 586.624,A 0.000,B 0.000,C 90.000,E1 112.333} C_DIS
LIN {X -0.012,Y -380.815,Z 586.611,A 0.000,B 0.000,C 90.000,E1 109.993} C_DIS
LIN {X 0.019,Y -396.659,Z 586.598,A 0.000,B 0.000,C 90.000,E1 107.692} C_DIS
LIN {X 0.218,Y -414.065,Z 586.586,A 0.000,B 0.000,C 90.000,E1 105.426} C_DIS
LIN {X -0.162,Y -433.142,Z 586.574,A 0.000,B 0.000,C 90.000,E1 103.300} C_DIS
LIN {X -0.054,Y -453.277,Z 586.562,A 0.000,B 0.000,C 90.000,E1 101.243} C_DIS
LIN {X -0.122,Y -473.883,Z 586.552,A 0.000,B 0.000,C 90.000,E1 99.378} C_DIS
LIN {X -0.106,Y -475.865,Z 586.551,A 0.000,B 0.000,C 90.000,E1 99.151} C_DIS
LIN {X 0.228,Y -477.549,Z 586.549,A 0.000,B 0.000,C 90.000,E1 98.859} C_DIS
LIN {X 0.090,Y -478.813,Z 586.548,A 0.000,B 0.000,C 90.000,E1 98.624} C_DIS
LIN {X 0.236,Y -480.375,Z 586.545,A 0.000,B 0.000,C 90.000,E1 98.106} C_DIS
LIN {X -0.087,Y -480.884,Z 586.542,A 0.000,B 0.000,C 90.000,E1 97.644} C_DIS
LIN {X 0.079,Y -480.421,Z 586.540,A 0.000,B 0.000,C 90.000,E1 97.125} C_DIS
LIN {X -0.229,Y -478.917,Z 586.537,A 0.000,B 0.000,C 90.000,E1 96.663} C_DIS
LIN {X 0.118,Y -477.695,Z 586.535,A 0.000,B 0.000,C 90.000,E1 96.372} C_DIS
LIN {X -0.064,Y -476.067,Z 586.534,A 0.000,B 0.000,C 90.000,E1 96.144} C_DIS
LIN {X 0.166,Y -459.460,Z 586.521,A 0.000,B 0.000,C 90.000,E1 93.841} C_DIS
LIN {X 0.184,Y -449.562,Z 586.513,A 0.000,B 0.000,C 90.000,E1 92.293} C_DIS
LIN {X -0.144,Y -434.940,Z 586.498,A 0.000,B 0.000,C 90.000,E1 89.714} C_DIS
LIN {X 0.180,Y -427.309,Z 586.491,A 0.000,B 0.000,C 90.000,E1 88.339} C_DIS
LIN {X 0.201,Y -416.154,Z 586.480,A 0.000,B 0.000,C 90.000,E1 86.445} C_DIS
LIN {X -0.167,Y -400.557,Z 586.465,A 0.000,B 0.000,C 90.000,E1 83.742} C_DIS
LIN {X -0.146,Y -388.628,Z 586.453,A 0.000,B 0.000,C 90.000,E1 81.489} C_DIS
LIN {X 0.085,Y -376.931,Z 586.440,A 0.000,B 0.000,C 90.000,E1 79.162} C_DIS
LIN {X 0.079,Y -364.096,Z 586.425,A 0.000,B 0.000,C 90.000,E1 76.533} C_DIS
LIN {X 0.009,Y -350.701,Z 586.409,A 0.000,B 0.000,C 90.000,E1 73.559} C_DIS
LIN {X 0.079,Y -337.531,Z 586.390,A 0.000,B 0.000,C 90.000,E1 70.188} C_DIS
LIN {X -0.185,Y -323.890,Z 586.367,A 0.000,B 0.000,C 90.000,E1 66.177} C_DIS
LIN {X 0.078,Y -316.219,Z 586.353,A 0.000,B 0.000,C 90.000,E1 63.589} C_DIS
LIN {X -0.132,Y -308.756,Z 586.339,A 0.000,B 0.000,C 90.000,E1 61.051} C_DIS
LIN {X 0.049,Y -301.492,Z 586.325,A 0.000,B 0.000,C 90.000,E1 58.408} C_DIS
LIN {X 0.023,Y -292.745,Z 586.306,A 0.000,B 0.000,C 90.000,E1 55.102} C_DIS
LIN {X -0.056,Y -286.160,Z 586.291,A 0.000,B 0.000,C 90.000,E1 52.431} C_DIS
LIN {X 0.139,Y -281.152,Z 586.280,A 0.000,B 0.000,C 90.000,E1 50.356} C_DIS
LIN {X 0.025,Y -275.767,Z 586.268,A 0.000,B 0.000,C 90.000,E1 48.324} C_DIS
LIN {X 0.014,Y -271.880,Z 586.261,A 0.000,B 0.000,C 90.000,E1 46.944} C_DIS
LIN {X 0.016,Y -266.554,Z 586.251,A 0.000,B 0.000,C 90.000,E1 45.202} C_DIS
LIN {X 0.008,Y -258.556,Z 586.237,A 0.000,B 0.000,C 90.000,E1 42.732} C_DIS
LIN {X 0.073,Y -247.195,Z 586.217,A 0.000,B 0.000,C 90.000,E1 39.116} C_DIS
LIN {X -0.072,Y -238.930,Z 586.201,A 0.000,B 0.000,C 90.000,E1 36.217} C_DIS
LIN {X 0.021,Y -231.318,Z 586.185,A 0.000,B 0.000,C 90.000,E1 33.214} C_DIS
LIN {X -0.059,Y -224.396,Z 586.168,A 0.000,B 0.000,C 90.000,E1 30.207} C_DIS
LIN {X -0.028,Y -218.197,Z 586.151,A 0.000,B 0.000,C 90.000,E1 27.129} C_DIS
LIN {X 0.081,Y -211.523,Z 586.129,A 0.000,B 0.000,C 90.000,E1 23.206} C_DIS
LIN {X 0.028,Y -207.097,Z 586.112,A 0.000,B 0.000,C 90.000,E1 20.066} C_DIS
LIN {X 0.041,Y -202.674,Z 586.089,A 0.000,B 0.000,C 90.000,E1 16.079} C_DIS
LIN {X 0.070,Y -198.740,Z 586.063,A 0.000,B 0.000,C 90.000,E1 11.243} C_DIS
LIN {X 0.053,Y -196.074,Z 586.031,A 0.000,B 0.000,C 90.000,E1 5.568} C_DIS
LIN {X 0.100,Y -197.278,Z 585.966,A 0.000,B 0.000,C 90.000,E1 353.799} C_DIS
LIN {X -0.076,Y -200.212,Z 585.939,A 0.000,B 0.000,C 90.000,E1 348.982} C_DIS
LIN {X -0.100,Y -204.533,Z 585.912,A 0.000,B 0.000,C 90.000,E1 344.157} C_DIS
LIN {X 0.017,Y -208.906,Z 585.890,A 0.000,B 0.000,C 90.000,E1 340.134} C_DIS
LIN {X 0.040,Y -214.150,Z 585.868,A 0.000,B 0.000,C 90.000,E1 336.177} C_DIS
LIN {X 0.002,Y -220.065,Z 585.846,A 0.000,B 0.000,C 90.000,E1 332.281} C_DIS
LIN {X 0.072,Y -226.558,Z 585.825,A 0.000,B 0.000,C 90.000,E1 328.408} C_DIS
LIN {X 0.055,Y -233.597,Z 585.803,A 0.000,B 0.000,C 90.000,E1 324.609} C_DIS
LIN {X -0.041,Y -241.039,Z 585.783,A 0.000,B 0.000,C 90.000,E1 320.884} C_DIS
LIN {X -0.015,Y -249.223,Z 585.762,A 0.000,B 0.000,C 90.000,E1 317.187} C_DIS
LIN {X 0.054,Y -258.346,Z 585.742,A 0.000,B 0.000,C 90.000,E1 313.542} C_DIS
LIN {X 0.062,Y -267.710,Z 585.724,A 0.000,B 0.000,C 90.000,E1 310.334} C_DIS
LIN {X 0.125,Y -277.373,Z 585.709,A 0.000,B 0.000,C 90.000,E1 307.523} C_DIS
LIN {X 0.028,Y -290.772,Z 585.690,A 0.000,B 0.000,C 90.000,E1 304.119} C_DIS
LIN {X -0.052,Y -305.738,Z 585.671,A 0.000,B 0.000,C 90.000,E1 300.797} C_DIS
LIN {X 0.073,Y -320.151,Z 585.655,A 0.000,B 0.000,C 90.000,E1 297.847} C_DIS
LIN {X -0.116,Y -335.569,Z 585.639,A 0.000,B 0.000,C 90.000,E1 295.027} C_DIS
LIN {X 0.132,Y -350.619,Z 585.625,A 0.000,B 0.000,C 90.000,E1 292.514} C_DIS
LIN {X 0.040,Y -367.165,Z 585.612,A 0.000,B 0.000,C 90.000,E1 290.120} C_DIS
LIN {X 0.122,Y -385.163,Z 585.599,A 0.000,B 0.000,C 90.000,E1 287.764} C_DIS
LIN {X -0.077,Y -399.372,Z 585.589,A 0.000,B 0.000,C 90.000,E1 286.079} C_DIS
LIN {X -0.148,Y -413.446,Z 585.580,A 0.000,B 0.000,C 90.000,E1 284.411} C_DIS
LIN {X 0.090,Y -425.165,Z 585.572,A 0.000,B 0.000,C 90.000,E1 283.008} C_DIS
LIN {X -0.081,Y -434.147,Z 585.566,A 0.000,B 0.000,C 90.000,E1 281.951} C_DIS
LIN {X -0.152,Y -442.582,Z 585.560,A 0.000,B 0.000,C 90.000,E1 280.894} C_DIS
LIN {X 0.035,Y -452.552,Z 585.553,A 0.000,B 0.000,C 90.000,E1 279.557} C_DIS
LIN {X 0.099,Y -459.819,Z 585.547,A 0.000,B 0.000,C 90.000,E1 278.511} C_DIS
LIN {X 0.185,Y -466.560,Z 585.542,A 0.000,B 0.000,C 90.000,E1 277.473} C_DIS
LIN {X 0.098,Y -471.240,Z 585.537,A 0.000,B 0.000,C 90.000,E1 276.720} C_DIS
LIN {X 0.049,Y -475.479,Z 585.533,A 0.000,B 0.000,C 90.000,E1 275.967} C_DIS
LIN {X -0.017,Y -479.117,Z 585.529,A 0.000,B 0.000,C 90.000,E1 275.220} C_DIS
LIN {X 0.131,Y -481.122,Z 585.526,A 0.000,B 0.000,C 90.000,E1 274.702} C_DIS
LIN {X -0.232,Y -482.812,Z 585.523,A 0.000,B 0.000,C 90.000,E1 274.245} C_DIS
LIN {X -0.065,Y -484.214,Z 585.521,A 0.000,B 0.000,C 90.000,E1 273.726} C_DIS
LIN {X 0.081,Y -485.349,Z 585.518,A 0.000,B 0.000,C 90.000,E1 273.212} C_DIS
LIN {X -0.223,Y -486.160,Z 585.515,A 0.000,B 0.000,C 90.000,E1 272.751} C_DIS
LIN {X -0.059,Y -486.657,Z 585.512,A 0.000,B 0.000,C 90.000,E1 272.236} C_DIS
LIN {X 0.128,Y -486.732,Z 585.510,A 0.000,B 0.000,C 90.000,E1 271.718} C_DIS
LIN {X -0.186,Y -486.327,Z 585.507,A 0.000,B 0.000,C 90.000,E1 271.260} C_DIS
LIN {X -0.011,Y -485.499,Z 585.504,A 0.000,B 0.000,C 90.000,E1 270.745} C_DIS
LIN {X 0.162,Y -484.074,Z 585.501,A 0.000,B 0.000,C 90.000,E1 270.229} C_DIS
LIN {X -0.154,Y -482.085,Z 585.499,A 0.000,B 0.000,C 90.000,E1 269.771} C_DIS
LIN {X 0.006,Y -479.348,Z 585.496,A 0.000,B 0.000,C 90.000,E1 269.255} C_DIS
LIN {X 0.144,Y -475.746,Z 585.493,A 0.000,B 0.000,C 90.000,E1 268.740} C_DIS
LIN {X -0.211,Y -471.116,Z 585.490,A 0.000,B 0.000,C 90.000,E1 268.282} C_DIS
LIN {X 0.095,Y -468.349,Z 585.489,A 0.000,B 0.000,C 90.000,E1 267.993} C_DIS
LIN {X -0.083,Y -465.253,Z 585.488,A 0.000,B 0.000,C 90.000,E1 267.764} C_DIS
LIN {X 0.020,Y -462.196,Z 585.486,A 0.000,B 0.000,C 90.000,E1 267.535} C_DIS
LIN {X 0.120,Y -458.673,Z 585.485,A 0.000,B 0.000,C 90.000,E1 267.306} C_DIS
LIN {X 0.045,Y -451.904,Z 585.483,A 0.000,B 0.000,C 90.000,E1 266.963} C_DIS
LIN {X -0.072,Y -444.202,Z 585.481,A 0.000,B 0.000,C 90.000,E1 266.674} C_DIS
LIN {X -0.053,Y -436.514,Z 585.480,A 0.000,B 0.000,C 90.000,E1 266.445} C_DIS
LIN {X -0.048,Y -427.998,Z 585.479,A 0.000,B 0.000,C 90.000,E1 266.274} C_DIS
LIN {X -0.066,Y -418.383,Z 585.479,A 0.000,B 0.000,C 90.000,E1 266.159} C_DIS
LIN {X -0.083,Y -408.360,Z 585.478,A 0.000,B 0.000,C 90.000,E1 266.102} C_DIS
LIN {X -0.068,Y -180.923,Z 585.478,A 0.000,B 0.000,C 90.000,E1 266.102} C_DIS
LIN {X -0.023,Y -180.874,Z 585.473,A 0.000,B 0.000,C 90.000,E1 265.065} C_DIS
LIN {X 0.059,Y -178.939,Z 585.443,A 0.000,B 0.000,C 90.000,E1 259.803} C_DIS
LIN {X -0.074,Y -175.988,Z 585.415,A 0.000,B 0.000,C 90.000,E1 254.755} C_DIS
LIN {X 0.041,Y -175.487,Z 585.410,A 0.000,B 0.000,C 90.000,E1 253.866} C_DIS
LIN {X 0.097,Y -172.232,Z 585.387,A 0.000,B 0.000,C 90.000,E1 249.571} C_DIS
LIN {X 0.074,Y -171.710,Z 585.382,A 0.000,B 0.000,C 90.000,E1 248.720} C_DIS
LIN {X 0.000,Y -167.304,Z 585.353,A 0.000,B 0.000,C 90.000,E1 243.563} C_DIS
LIN {X 0.005,Y -166.684,Z 585.348,A 0.000,B 0.000,C 90.000,E1 242.692} C_DIS
LIN {X -0.003,Y -162.666,Z 585.324,A 0.000,B 0.000,C 90.000,E1 238.329} C_DIS
LIN {X -0.030,Y -161.355,Z 585.314,A 0.000,B 0.000,C 90.000,E1 236.580} C_DIS
LIN {X 0.004,Y -157.349,Z 585.290,A 0.000,B 0.000,C 90.000,E1 232.145} C_DIS
LIN {X 0.033,Y -155.336,Z 585.275,A 0.000,B 0.000,C 90.000,E1 229.461} C_DIS
LIN {X -0.037,Y -151.686,Z 585.250,A 0.000,B 0.000,C 90.000,E1 225.000} C_DIS
LIN {X 0.011,Y -150.549,Z 585.240,A 0.000,B 0.000,C 90.000,E1 223.176} C_DIS
LIN {X 0.043,Y -147.275,Z 585.215,A 0.000,B 0.000,C 90.000,E1 218.624} C_DIS
LIN {X 0.016,Y -145.302,Z 585.194,A 0.000,B 0.000,C 90.000,E1 214.978} C_DIS
LIN {X 0.008,Y -142.396,Z 585.164,A 0.000,B 0.000,C 90.000,E1 209.461} C_DIS
LIN {X -0.009,Y -141.376,Z 585.148,A 0.000,B 0.000,C 90.000,E1 206.693} C_DIS
LIN {X 0.032,Y -139.347,Z 585.112,A 0.000,B 0.000,C 90.000,E1 200.174} C_DIS
LIN {X -0.027,Y -138.784,Z 585.097,A 0.000,B 0.000,C 90.000,E1 197.402} C_DIS
LIN {X 0.032,Y -138.344,Z 585.055,A 0.000,B 0.000,C 90.000,E1 189.905} C_DIS
LIN {X 0.052,Y -139.389,Z 585.008,A 0.000,B 0.000,C 90.000,E1 181.489} C_DIS
LIN {X -0.034,Y -141.287,Z 584.972,A 0.000,B 0.000,C 90.000,E1 175.008} C_DIS
LIN {X 0.065,Y -142.651,Z 584.957,A 0.000,B 0.000,C 90.000,E1 172.186} C_DIS
LIN {X 0.015,Y -144.989,Z 584.931,A 0.000,B 0.000,C 90.000,E1 167.589} C_DIS
LIN {X 0.006,Y -147.616,Z 584.911,A 0.000,B 0.000,C 90.000,E1 163.921} C_DIS
LIN {X 0.084,Y -150.240,Z 584.890,A 0.000,B 0.000,C 90.000,E1 160.242} C_DIS
LIN {X -0.043,Y -153.633,Z 584.870,A 0.000,B 0.000,C 90.000,E1 156.666} C_DIS
LIN {X 0.016,Y -157.049,Z 584.850,A 0.000,B 0.000,C 90.000,E1 153.050} C_DIS
LIN {X 0.015,Y -161.177,Z 584.831,A 0.000,B 0.000,C 90.000,E1 149.488} C_DIS
LIN {X 0.044,Y -163.271,Z 584.821,A 0.000,B 0.000,C 90.000,E1 147.709} C_DIS
LIN {X 0.056,Y -167.712,Z 584.801,A 0.000,B 0.000,C 90.000,E1 144.196} C_DIS
LIN {X -0.032,Y -171.531,Z 584.787,A 0.000,B 0.000,C 90.000,E1 141.618} C_DIS
LIN {X 0.010,Y -176.472,Z 584.768,A 0.000,B 0.000,C 90.000,E1 138.162} C_DIS
LIN {X 0.010,Y -180.769,Z 584.753,A 0.000,B 0.000,C 90.000,E1 135.607} C_DIS
LIN {X -0.002,Y -186.175,Z 584.735,A 0.000,B 0.000,C 90.000,E1 132.243} C_DIS
LIN {X -0.014,Y -191.382,Z 584.719,A 0.000,B 0.000,C 90.000,E1 129.402} C_DIS
LIN {X 0.010,Y -191.443,Z 584.719,A 0.000,B 0.000,C 90.000,E1 129.358} C_DIS
LIN {X -0.028,Y -288.403,Z 584.719,A 0.000,B 0.000,C 90.000,E1 129.358} C_DIS
LIN {X -0.116,Y -289.776,Z 584.719,A 0.000,B 0.000,C 90.000,E1 129.358} C_DIS
LIN {X 0.050,Y -294.578,Z 584.717,A 0.000,B 0.000,C 90.000,E1 129.116} C_DIS
LIN {X 0.033,Y -297.079,Z 584.716,A 0.000,B 0.000,C 90.000,E1 128.910} C_DIS
LIN {X 0.038,Y -300.895,Z 584.714,A 0.000,B 0.000,C 90.000,E1 128.418} C_DIS
LIN {X -0.018,Y -302.688,Z 584.712,A 0.000,B 0.000,C 90.000,E1 128.096} C_DIS
LIN {X 0.164,Y -304.090,Z 584.710,A 0.000,B 0.000,C 90.000,E1 127.729} C_DIS
LIN {X -0.067,Y -307.928,Z 584.702,A 0.000,B 0.000,C 90.000,E1 126.457} C_DIS
LIN {X -0.095,Y -317.996,Z 584.684,A 0.000,B 0.000,C 90.000,E1 123.214} C_DIS
LIN {X -0.047,Y -328.377,Z 584.668,A 0.000,B 0.000,C 90.000,E1 120.335} C_DIS
LIN {X -0.025,Y -340.115,Z 584.653,A 0.000,B 0.000,C 90.000,E1 117.513} C_DIS
LIN {X -0.136,Y -353.309,Z 584.638,A 0.000,B 0.000,C 90.000,E1 114.771} C_DIS
LIN {X 0.087,Y -366.360,Z 584.624,A 0.000,B 0.000,C 90.000,E1 112.333} C_DIS
LIN {X 0.024,Y -380.754,Z 584.611,A 0.000,B 0.000,C 90.000,E1 109.993} C_DIS
LIN {X 0.056,Y -396.594,Z 584.598,A 0.000,B 0.000,C 90.000,E1 107.692} C_DIS
LIN {X -0.145,Y -413.997,Z 584.586,A 0.000,B 0.000,C 90.000,E1 105.481} C_DIS
LIN {X -0.125,Y -433.070,Z 584.574,A 0.000,B 0.000,C 90.000,E1 103.300} C_DIS
LIN {X -0.020,Y -453.203,Z 584.562,A 0.000,B 0.000,C 90.000,E1 101.243} C_DIS
LIN {X -0.091,Y -473.830,Z 584.552,A 0.000,B 0.000,C 90.000,E1 99.378} C_DIS
LIN {X -0.075,Y -475.856,Z 584.551,A 0.000,B 0.000,C 90.000,E1 99.151} C_DIS
LIN {X -0.213,Y -477.573,Z 584.549,A 0.000,B 0.000,C 90.000,E1 98.916} C_DIS
LIN {X 0.120,Y -478.862,Z 584.548,A 0.000,B 0.000,C 90.000,E1 98.624} C_DIS
LIN {X -0.210,Y -480.461,Z 584.545,A 0.000,B 0.000,C 90.000,E1 98.163} C_DIS
LIN {X -0.055,Y -481.000,Z 584.542,A 0.000,B 0.000,C 90.000,E1 97.644} C_DIS
LIN {X 0.111,Y -480.569,Z 584.540,A 0.000,B 0.000,C 90.000,E1 97.125} C_DIS
LIN {X -0.197,Y -479.100,Z 584.537,A 0.000,B 0.000,C 90.000,E1 96.663} C_DIS
LIN {X 0.150,Y -477.901,Z 584.536,A 0.000,B 0.000,C 90.000,E1 96.372} C_DIS
LIN {X -0.031,Y -476.302,Z 584.534,A 0.000,B 0.000,C 90.000,E1 96.144} C_DIS
LIN {X 0.204,Y -459.655,Z 584.521,A 0.000,B 0.000,C 90.000,E1 93.841} C_DIS
LIN {X -0.225,Y -449.715,Z 584.513,A 0.000,B 0.000,C 90.000,E1 92.350} C_DIS
LIN {X -0.102,Y -435.064,Z 584.498,A 0.000,B 0.000,C 90.000,E1 89.714} C_DIS
LIN {X -0.204,Y -427.432,Z 584.491,A 0.000,B 0.000,C 90.000,E1 88.396} C_DIS
LIN {X -0.170,Y -416.260,Z 584.480,A 0.000,B 0.000,C 90.000,E1 86.502} C_DIS
LIN {X -0.208,Y -402.184,Z 584.467,A 0.000,B 0.000,C 90.000,E1 84.033} C_DIS
LIN {X -0.099,Y -388.714,Z 584.453,A 0.000,B 0.000,C 90.000,E1 81.489} C_DIS
LIN {X 0.133,Y -376.994,Z 584.440,A 0.000,B 0.000,C 90.000,E1 79.162} C_DIS
LIN {X 0.126,Y -364.104,Z 584.425,A 0.000,B 0.000,C 90.000,E1 76.533} C_DIS
LIN {X 0.055,Y -350.702,Z 584.409,A 0.000,B 0.000,C 90.000,E1 73.559} C_DIS
LIN {X 0.123,Y -337.555,Z 584.390,A 0.000,B 0.000,C 90.000,E1 70.188} C_DIS
LIN {X -0.140,Y -323.950,Z 584.367,A 0.000,B 0.000,C 90.000,E1 66.177} C_DIS
LIN {X -0.161,Y -314.410,Z 584.350,A 0.000,B 0.000,C 90.000,E1 62.999} C_DIS
LIN {X 0.016,Y -307.016,Z 584.335,A 0.000,B 0.000,C 90.000,E1 60.383} C_DIS
LIN {X -0.105,Y -299.768,Z 584.321,A 0.000,B 0.000,C 90.000,E1 57.788} C_DIS
LIN {X -0.178,Y -291.141,Z 584.302,A 0.000,B 0.000,C 90.000,E1 54.482} C_DIS
LIN {X -0.008,Y -286.201,Z 584.291,A 0.000,B 0.000,C 90.000,E1 52.431} C_DIS
LIN {X 0.187,Y -281.179,Z 584.280,A 0.000,B 0.000,C 90.000,E1 50.356} C_DIS
LIN {X 0.061,Y -277.646,Z 584.272,A 0.000,B 0.000,C 90.000,E1 49.013} C_DIS
LIN {X 0.073,Y -273.872,Z 584.265,A 0.000,B 0.000,C 90.000,E1 47.634} C_DIS
LIN {X -0.158,Y -269.835,Z 584.257,A 0.000,B 0.000,C 90.000,E1 46.296} C_DIS
LIN {X 0.000,Y -264.299,Z 584.247,A 0.000,B 0.000,C 90.000,E1 44.514} C_DIS
LIN {X 0.093,Y -257.358,Z 584.235,A 0.000,B 0.000,C 90.000,E1 42.366} C_DIS
LIN {X 0.116,Y -247.175,Z 584.217,A 0.000,B 0.000,C 90.000,E1 39.116} C_DIS
LIN {X -0.031,Y -238.911,Z 584.201,A 0.000,B 0.000,C 90.000,E1 36.217} C_DIS
LIN {X -0.067,Y -231.298,Z 584.185,A 0.000,B 0.000,C 90.000,E1 33.245} C_DIS
LIN {X -0.023,Y -224.362,Z 584.168,A 0.000,B 0.000,C 90.000,E1 30.207} C_DIS
LIN {X 0.007,Y -218.170,Z 584.151,A 0.000,B 0.000,C 90.000,E1 27.129} C_DIS
LIN {X -0.023,Y -212.713,Z 584.133,A 0.000,B 0.000,C 90.000,E1 24.027} C_DIS
LIN {X 0.035,Y -208.044,Z 584.116,A 0.000,B 0.000,C 90.000,E1 20.865} C_DIS
LIN {X -0.052,Y -203.416,Z 584.094,A 0.000,B 0.000,C 90.000,E1 16.913} C_DIS
LIN {X 0.053,Y -199.260,Z 584.067,A 0.000,B 0.000,C 90.000,E1 12.063} C_DIS
LIN {X -0.084,Y -196.295,Z 584.036,A 0.000,B 0.000,C 90.000,E1 6.429} C_DIS
LIN {X 0.066,Y -197.642,Z 583.961,A 0.000,B 0.000,C 90.000,E1 352.996} C_DIS
LIN {X -0.074,Y -200.891,Z 583.934,A 0.000,B 0.000,C 90.000,E1 348.173} C_DIS
LIN {X 0.019,Y -205.353,Z 583.907,A 0.000,B 0.000,C 90.000,E1 343.323} C_DIS
LIN {X 0.032,Y -209.929,Z 583.885,A 0.000,B 0.000,C 90.000,E1 339.337} C_DIS
LIN {X -0.022,Y -215.295,Z 583.863,A 0.000,B 0.000,C 90.000,E1 335.409} C_DIS
LIN {X -0.023,Y -221.318,Z 583.842,A 0.000,B 0.000,C 90.000,E1 331.513} C_DIS
LIN {X 0.001,Y -227.919,Z 583.820,A 0.000,B 0.000,C 90.000,E1 327.661} C_DIS
LIN {X 0.056,Y -233.591,Z 583.803,A 0.000,B 0.000,C 90.000,E1 324.609} C_DIS
LIN {X -0.039,Y -241.020,Z 583.783,A 0.000,B 0.000,C 90.000,E1 320.884} C_DIS
LIN {X -0.015,Y -249.201,Z 583.762,A 0.000,B 0.000,C 90.000,E1 317.187} C_DIS
LIN {X 0.054,Y -258.316,Z 583.742,A 0.000,B 0.000,C 90.000,E1 313.542} C_DIS
LIN {X 0.061,Y -267.677,Z 583.724,A 0.000,B 0.000,C 90.000,E1 310.334} C_DIS
LIN {X 0.000,Y -278.623,Z 583.707,A 0.000,B 0.000,C 90.000,E1 307.202} C_DIS
LIN {X 0.026,Y -290.739,Z 583.690,A 0.000,B 0.000,C 90.000,E1 304.119} C_DIS
LIN {X -0.057,Y -305.676,Z 583.671,A 0.000,B 0.000,C 90.000,E1 300.797} C_DIS
LIN {X 0.067,Y -320.052,Z 583.655,A 0.000,B 0.000,C 90.000,E1 297.847} C_DIS
LIN {X -0.125,Y -335.463,Z 583.639,A 0.000,B 0.000,C 90.000,E1 295.027} C_DIS
LIN {X 0.119,Y -350.526,Z 583.625,A 0.000,B 0.000,C 90.000,E1 292.514} C_DIS
LIN {X 0.027,Y -367.118,Z 583.612,A 0.000,B 0.000,C 90.000,E1 290.120} C_DIS
LIN {X 0.107,Y -385.137,Z 583.599,A 0.000,B 0.000,C 90.000,E1 287.764} C_DIS
LIN {X -0.093,Y -399.362,Z 583.589,A 0.000,B 0.000,C 90.000,E1 286.079} C_DIS
LIN {X -0.148,Y -413.461,Z 583.580,A 0.000,B 0.000,C 90.000,E1 284.411} C_DIS
LIN {X 0.107,Y -425.184,Z 583.572,A 0.000,B 0.000,C 90.000,E1 283.008} C_DIS
LIN {X -0.064,Y -434.180,Z 583.566,A 0.000,B 0.000,C 90.000,E1 281.951} C_DIS
LIN {X -0.133,Y -442.629,Z 583.560,A 0.000,B 0.000,C 90.000,E1 280.894} C_DIS
LIN {X -0.190,Y -450.689,Z 583.555,A 0.000,B 0.000,C 90.000,E1 279.849} C_DIS
LIN {X -0.152,Y -458.109,Z 583.549,A 0.000,B 0.000,C 90.000,E1 278.803} C_DIS
LIN {X -0.026,Y -464.961,Z 583.543,A 0.000,B 0.000,C 90.000,E1 277.757} C_DIS
LIN {X 0.119,Y -471.276,Z 583.537,A 0.000,B 0.000,C 90.000,E1 276.720} C_DIS
LIN {X 0.072,Y -475.476,Z 583.533,A 0.000,B 0.000,C 90.000,E1 275.967} C_DIS
LIN {X 0.004,Y -479.113,Z 583.529,A 0.000,B 0.000,C 90.000,E1 275.220} C_DIS
LIN {X 0.153,Y -481.128,Z 583.526,A 0.000,B 0.000,C 90.000,E1 274.702} C_DIS
LIN {X -0.209,Y -482.807,Z 583.523,A 0.000,B 0.000,C 90.000,E1 274.245} C_DIS
LIN {X -0.043,Y -484.235,Z 583.521,A 0.000,B 0.000,C 90.000,E1 273.726} C_DIS
LIN {X 0.103,Y -485.392,Z 583.518,A 0.000,B 0.000,C 90.000,E1 273.212} C_DIS
LIN {X -0.201,Y -486.253,Z 583.515,A 0.000,B 0.000,C 90.000,E1 272.751} C_DIS
LIN {X -0.036,Y -486.730,Z 583.512,A 0.000,B 0.000,C 90.000,E1 272.236} C_DIS
LIN {X 0.152,Y -486.831,Z 583.510,A 0.000,B 0.000,C 90.000,E1 271.718} C_DIS
LIN {X -0.162,Y -486.435,Z 583.507,A 0.000,B 0.000,C 90.000,E1 271.260} C_DIS
LIN {X 0.013,Y -485.561,Z 583.504,A 0.000,B 0.000,C 90.000,E1 270.745} C_DIS
LIN {X 0.187,Y -484.103,Z 583.501,A 0.000,B 0.000,C 90.000,E1 270.229} C_DIS
LIN {X -0.128,Y -482.064,Z 583.499,A 0.000,B 0.000,C 90.000,E1 269.771} C_DIS
LIN {X 0.031,Y -479.336,Z 583.496,A 0.000,B 0.000,C 90.000,E1 269.255} C_DIS
LIN {X -0.139,Y -477.679,Z 583.495,A 0.000,B 0.000,C 90.000,E1 269.026} C_DIS
LIN {X -0.009,Y -473.565,Z 583.492,A 0.000,B 0.000,C 90.000,E1 268.511} C_DIS
LIN {X 0.127,Y -468.377,Z 583.489,A 0.000,B 0.000,C 90.000,E1 267.993} C_DIS
LIN {X 0.085,Y -462.274,Z 583.486,A 0.000,B 0.000,C 90.000,E1 267.535} C_DIS
LIN {X 0.154,Y -455.605,Z 583.484,A 0.000,B 0.000,C 90.000,E1 267.135} C_DIS
LIN {X -0.136,Y -448.557,Z 583.482,A 0.000,B 0.000,C 90.000,E1 266.846} C_DIS
LIN {X 0.049,Y -441.076,Z 583.481,A 0.000,B 0.000,C 90.000,E1 266.560} C_DIS
LIN {X -0.196,Y -433.044,Z 583.480,A 0.000,B 0.000,C 90.000,E1 266.388} C_DIS
LIN {X -0.026,Y -424.289,Z 583.479,A 0.000,B 0.000,C 90.000,E1 266.216} C_DIS
LIN {X 0.069,Y -413.801,Z 583.478,A 0.000,B 0.000,C 90.000,E1 266.102} C_DIS
LIN {X -0.077,Y -409.275,Z 583.478,A 0.000,B 0.000,C 90.000,E1 266.102} C_DIS
LIN {X -0.066,Y -180.924,Z 583.478,A 0.000,B 0.000,C 90.000,E1 266.102} C_DIS
LIN {X -0.022,Y -180.874,Z 583.473,A 0.000,B 0.000,C 90.000,E1 265.065} C_DIS
LIN {X 0.061,Y -178.939,Z 583.443,A 0.000,B 0.000,C 90.000,E1 259.803} C_DIS
LIN {X -0.072,Y -175.989,Z 583.415,A 0.000,B 0.000,C 90.000,E1 254.755} C_DIS
LIN {X 0.043,Y -175.488,Z 583.410,A 0.000,B 0.000,C 90.000,E1 253.866} C_DIS
LIN {X 0.099,Y -172.232,Z 583.387,A 0.000,B 0.000,C 90.000,E1 249.571} C_DIS
LIN {X 0.077,Y -171.710,Z 583.382,A 0.000,B 0.000,C 90.000,E1 248.720} C_DIS
LIN {X 0.001,Y -167.304,Z 583.353,A 0.000,B 0.000,C 90.000,E1 243.563} C_DIS
LIN {X 0.006,Y -166.684,Z 583.348,A 0.000,B 0.000,C 90.000,E1 242.692} C_DIS
LIN {X -0.002,Y -162.666,Z 583.324,A 0.000,B 0.000,C 90.000,E1 238.329} C_DIS
LIN {X -0.029,Y -161.355,Z 583.314,A 0.000,B 0.000,C 90.000,E1 236.580} C_DIS
LIN {X 0.006,Y -157.349,Z 583.290,A 0.000,B 0.000,C 90.000,E1 232.145} C_DIS
LIN {X 0.034,Y -155.337,Z 583.275,A 0.000,B 0.000,C 90.000,E1 229.461} C_DIS
LIN {X -0.035,Y -151.686,Z 583.250,A 0.000,B 0.000,C 90.000,E1 225.000} C_DIS
LIN {X 0.013,Y -150.549,Z 583.240,A 0.000,B 0.000,C 90.000,E1 223.176} C_DIS
LIN {X 0.045,Y -147.275,Z 583.215,A 0.000,B 0.000,C 90.000,E1 218.624} C_DIS
LIN {X 0.018,Y -145.303,Z 583.194,A 0.000,B 0.000,C 90.000,E1 214.978} C_DIS
LIN {X 0.009,Y -142.396,Z 583.164,A 0.000,B 0.000,C 90.000,E1 209.461} C_DIS
LIN {X -0.008,Y -141.377,Z 583.148,A 0.000,B 0.000,C 90.000,E1 206.693} C_DIS
LIN {X 0.033,Y -139.347,Z 583.112,A 0.000,B 0.000,C 90.000,E1 200.174} C_DIS
LIN {X -0.024,Y -138.784,Z 583.097,A 0.000,B 0.000,C 90.000,E1 197.402} C_DIS
LIN {X 0.034,Y -138.344,Z 583.055,A 0.000,B 0.000,C 90.000,E1 189.905} C_DIS
LIN {X 0.054,Y -139.389,Z 583.008,A 0.000,B 0.000,C 90.000,E1 181.489} C_DIS
LIN {X -0.033,Y -141.287,Z 582.972,A 0.000,B 0.000,C 90.000,E1 175.008} C_DIS
LIN {X 0.067,Y -142.651,Z 582.957,A 0.000,B 0.000,C 90.000,E1 172.186} C_DIS
LIN {X 0.016,Y -144.989,Z 582.931,A 0.000,B 0.000,C 90.000,E1 167.589} C_DIS
LIN {X 0.007,Y -147.616,Z 582.911,A 0.000,B 0.000,C 90.000,E1 163.921} C_DIS
LIN {X 0.085,Y -150.240,Z 582.890,A 0.000,B 0.000,C 90.000,E1 160.242} C_DIS
LIN {X -0.041,Y -153.633,Z 582.870,A 0.000,B 0.000,C 90.000,E1 156.666} C_DIS
LIN {X 0.017,Y -157.049,Z 582.850,A 0.000,B 0.000,C 90.000,E1 153.050} C_DIS
LIN {X 0.015,Y -161.176,Z 582.831,A 0.000,B 0.000,C 90.000,E1 149.488} C_DIS
LIN {X 0.046,Y -163.271,Z 582.821,A 0.000,B 0.000,C 90.000,E1 147.709} C_DIS
LIN {X 0.057,Y -167.712,Z 582.801,A 0.000,B 0.000,C 90.000,E1 144.196} C_DIS
LIN {X -0.030,Y -171.532,Z 582.787,A 0.000,B 0.000,C 90.000,E1 141.618} C_DIS
LIN {X 0.013,Y -176.471,Z 582.768,A 0.000,B 0.000,C 90.000,E1 138.162} C_DIS
LIN {X 0.011,Y -180.768,Z 582.753,A 0.000,B 0.000,C 90.000,E1 135.607} C_DIS
LIN {X 0.000,Y -186.174,Z 582.735,A 0.000,B 0.000,C 90.000,E1 132.243} C_DIS
LIN {X -0.013,Y -191.382,Z 582.719,A 0.000,B 0.000,C 90.000,E1 129.402} C_DIS
LIN {X -0.047,Y -191.471,Z 582.719,A 0.000,B 0.000,C 90.000,E1 129.358} C_DIS
LIN {X -0.115,Y -288.736,Z 582.719,A 0.000,B 0.000,C 90.000,E1 129.358} C_DIS
LIN {X 0.052,Y -294.374,Z 582.717,A 0.000,B 0.000,C 90.000,E1 129.116} C_DIS
LIN {X 0.035,Y -296.944,Z 582.716,A 0.000,B 0.000,C 90.000,E1 128.910} C_DIS
LIN {X -0.135,Y -300.751,Z 582.714,A 0.000,B 0.000,C 90.000,E1 128.463} C_DIS
LIN {X 0.045,Y -302.582,Z 582.712,A 0.000,B 0.000,C 90.000,E1 128.096} C_DIS
LIN {X -0.200,Y -304.011,Z 582.710,A 0.000,B 0.000,C 90.000,E1 127.810} C_DIS
LIN {X 0.013,Y -306.039,Z 582.706,A 0.000,B 0.000,C 90.000,E1 127.111} C_DIS
LIN {X -0.064,Y -315.802,Z 582.688,A 0.000,B 0.000,C 90.000,E1 123.865} C_DIS
LIN {X -0.175,Y -325.888,Z 582.672,A 0.000,B 0.000,C 90.000,E1 121.003} C_DIS
LIN {X -0.066,Y -337.311,Z 582.656,A 0.000,B 0.000,C 90.000,E1 118.153} C_DIS
LIN {X 0.205,Y -350.164,Z 582.641,A 0.000,B 0.000,C 90.000,E1 115.335} C_DIS
LIN {X 0.023,Y -362.889,Z 582.628,A 0.000,B 0.000,C 90.000,E1 112.950} C_DIS
LIN {X -0.129,Y -376.931,Z 582.614,A 0.000,B 0.000,C 90.000,E1 110.610} C_DIS
LIN {X -0.070,Y -392.392,Z 582.602,A 0.000,B 0.000,C 90.000,E1 108.290} C_DIS
LIN {X 0.011,Y -409.384,Z 582.589,A 0.000,B 0.000,C 90.000,E1 106.024} C_DIS
LIN {X 0.018,Y -428.033,Z 582.577,A 0.000,B 0.000,C 90.000,E1 103.828} C_DIS
LIN {X -0.215,Y -447.996,Z 582.565,A 0.000,B 0.000,C 90.000,E1 101.771} C_DIS
LIN {X -0.169,Y -468.542,Z 582.555,A 0.000,B 0.000,C 90.000,E1 99.849} C_DIS
LIN {X -0.026,Y -473.731,Z 582.552,A 0.000,B 0.000,C 90.000,E1 99.378} C_DIS
LIN {X -0.011,Y -475.810,Z 582.551,A 0.000,B 0.000,C 90.000,E1 99.151} C_DIS
LIN {X -0.148,Y -477.567,Z 582.549,A 0.000,B 0.000,C 90.000,E1 98.916} C_DIS
LIN {X 0.185,Y -478.887,Z 582.548,A 0.000,B 0.000,C 90.000,E1 98.624} C_DIS
LIN {X -0.145,Y -480.533,Z 582.545,A 0.000,B 0.000,C 90.000,E1 98.163} C_DIS
LIN {X 0.010,Y -481.112,Z 582.542,A 0.000,B 0.000,C 90.000,E1 97.644} C_DIS
LIN {X 0.175,Y -480.720,Z 582.540,A 0.000,B 0.000,C 90.000,E1 97.125} C_DIS
LIN {X -0.131,Y -479.296,Z 582.537,A 0.000,B 0.000,C 90.000,E1 96.663} C_DIS
LIN {X 0.217,Y -478.125,Z 582.536,A 0.000,B 0.000,C 90.000,E1 96.372} C_DIS
LIN {X 0.036,Y -476.561,Z 582.534,A 0.000,B 0.000,C 90.000,E1 96.144} C_DIS
LIN {X -0.185,Y -459.871,Z 582.522,A 0.000,B 0.000,C 90.000,E1 93.898} C_DIS
LIN {X -0.154,Y -449.900,Z 582.513,A 0.000,B 0.000,C 90.000,E1 92.350} C_DIS
LIN {X -0.028,Y -435.217,Z 582.498,A 0.000,B 0.000,C 90.000,E1 89.714} C_DIS
LIN {X -0.128,Y -427.585,Z 582.491,A 0.000,B 0.000,C 90.000,E1 88.396} C_DIS
LIN {X -0.093,Y -416.391,Z 582.480,A 0.000,B 0.000,C 90.000,E1 86.502} C_DIS
LIN {X -0.185,Y -403.857,Z 582.468,A 0.000,B 0.000,C 90.000,E1 84.318} C_DIS
LIN {X -0.083,Y -391.780,Z 582.456,A 0.000,B 0.000,C 90.000,E1 82.064} C_DIS
LIN {X 0.164,Y -379.997,Z 582.443,A 0.000,B 0.000,C 90.000,E1 79.746} C_DIS
LIN {X -0.113,Y -368.395,Z 582.430,A 0.000,B 0.000,C 90.000,E1 77.465} C_DIS
LIN {X 0.095,Y -351.984,Z 582.410,A 0.000,B 0.000,C 90.000,E1 73.866} C_DIS
LIN {X -0.121,Y -337.593,Z 582.390,A 0.000,B 0.000,C 90.000,E1 70.242} C_DIS
LIN {X -0.068,Y -324.019,Z 582.368,A 0.000,B 0.000,C 90.000,E1 66.177} C_DIS
LIN {X -0.088,Y -314.506,Z 582.350,A 0.000,B 0.000,C 90.000,E1 62.999} C_DIS
LIN {X 0.089,Y -307.109,Z 582.336,A 0.000,B 0.000,C 90.000,E1 60.383} C_DIS
LIN {X -0.031,Y -299.850,Z 582.321,A 0.000,B 0.000,C 90.000,E1 57.788} C_DIS
LIN {X -0.104,Y -291.210,Z 582.303,A 0.000,B 0.000,C 90.000,E1 54.482} C_DIS
LIN {X -0.051,Y -284.590,Z 582.288,A 0.000,B 0.000,C 90.000,E1 51.778} C_DIS
LIN {X -0.101,Y -279.494,Z 582.276,A 0.000,B 0.000,C 90.000,E1 49.747} C_DIS
LIN {X -0.056,Y -273.899,Z 582.265,A 0.000,B 0.000,C 90.000,E1 47.676} C_DIS
LIN {X -0.086,Y -269.840,Z 582.257,A 0.000,B 0.000,C 90.000,E1 46.296} C_DIS
LIN {X 0.071,Y -264.294,Z 582.247,A 0.000,B 0.000,C 90.000,E1 44.514} C_DIS
LIN {X 0.013,Y -256.204,Z 582.234,A 0.000,B 0.000,C 90.000,E1 42.043} C_DIS
LIN {X 0.027,Y -247.170,Z 582.218,A 0.000,B 0.000,C 90.000,E1 39.152} C_DIS
LIN {X 0.033,Y -238.888,Z 582.201,A 0.000,B 0.000,C 90.000,E1 36.217} C_DIS
LIN {X -0.005,Y -231.291,Z 582.185,A 0.000,B 0.000,C 90.000,E1 33.245} C_DIS
LIN {X 0.037,Y -224.340,Z 582.168,A 0.000,B 0.000,C 90.000,E1 30.207} C_DIS
LIN {X 0.064,Y -218.135,Z 582.151,A 0.000,B 0.000,C 90.000,E1 27.129} C_DIS
LIN {X -0.026,Y -211.390,Z 582.129,A 0.000,B 0.000,C 90.000,E1 23.259} C_DIS
LIN {X -0.084,Y -206.956,Z 582.112,A 0.000,B 0.000,C 90.000,E1 20.120} C_DIS
LIN {X -0.078,Y -202.584,Z 582.090,A 0.000,B 0.000,C 90.000,E1 16.134} C_DIS
LIN {X -0.052,Y -198.665,Z 582.063,A 0.000,B 0.000,C 90.000,E1 11.299} C_DIS
LIN {X 0.103,Y -195.835,Z 582.027,A 0.000,B 0.000,C 90.000,E1 4.759} C_DIS
LIN {X 0.099,Y -197.240,Z 581.966,A 0.000,B 0.000,C 90.000,E1 353.799} C_DIS
LIN {X -0.077,Y -200.243,Z 581.939,A 0.000,B 0.000,C 90.000,E1 348.982} C_DIS
LIN {X -0.100,Y -204.561,Z 581.912,A 0.000,B 0.000,C 90.000,E1 344.157} C_DIS
LIN {X 0.017,Y -208.948,Z 581.890,A 0.000,B 0.000,C 90.000,E1 340.134} C_DIS
LIN {X 0.042,Y -214.196,Z 581.868,A 0.000,B 0.000,C 90.000,E1 336.177} C_DIS
LIN {X 0.005,Y -220.069,Z 581.846,A 0.000,B 0.000,C 90.000,E1 332.281} C_DIS
LIN {X 0.074,Y -226.553,Z 581.825,A 0.000,B 0.000,C 90.000,E1 328.408} C_DIS
LIN {X 0.057,Y -233.586,Z 581.803,A 0.000,B 0.000,C 90.000,E1 324.609} C_DIS
LIN {X -0.039,Y -241.002,Z 581.783,A 0.000,B 0.000,C 90.000,E1 320.884} C_DIS
LIN {X -0.014,Y -249.171,Z 581.762,A 0.000,B 0.000,C 90.000,E1 317.187} C_DIS
LIN {X 0.053,Y -258.287,Z 581.742,A 0.000,B 0.000,C 90.000,E1 313.542} C_DIS
LIN {X 0.059,Y -267.664,Z 581.724,A 0.000,B 0.000,C 90.000,E1 310.334} C_DIS
LIN {X -0.002,Y -278.613,Z 581.707,A 0.000,B 0.000,C 90.000,E1 307.202} C_DIS
LIN {X 0.023,Y -290.705,Z 581.690,A 0.000,B 0.000,C 90.000,E1 304.119} C_DIS
LIN {X -0.062,Y -305.611,Z 581.671,A 0.000,B 0.000,C 90.000,E1 300.797} C_DIS
LIN {X 0.060,Y -319.953,Z 581.655,A 0.000,B 0.000,C 90.000,E1 297.847} C_DIS
LIN {X -0.135,Y -335.366,Z 581.639,A 0.000,B 0.000,C 90.000,E1 295.027} C_DIS
LIN {X 0.106,Y -350.439,Z 581.625,A 0.000,B 0.000,C 90.000,E1 292.514} C_DIS
LIN {X 0.115,Y -366.950,Z 581.612,A 0.000,B 0.000,C 90.000,E1 290.120} C_DIS
LIN {X -0.171,Y -384.995,Z 581.599,A 0.000,B 0.000,C 90.000,E1 287.819} C_DIS
LIN {X 0.119,Y -399.084,Z 581.589,A 0.000,B 0.000,C 90.000,E1 286.079} C_DIS
LIN {X 0.051,Y -413.250,Z 581.580,A 0.000,B 0.000,C 90.000,E1 284.411} C_DIS
LIN {X 0.034,Y -427.329,Z 581.571,A 0.000,B 0.000,C 90.000,E1 282.771} C_DIS
LIN {X -0.114,Y -436.211,Z 581.565,A 0.000,B 0.000,C 90.000,E1 281.715} C_DIS
LIN {X 0.054,Y -446.601,Z 581.558,A 0.000,B 0.000,C 90.000,E1 280.366} C_DIS
LIN {X 0.045,Y -454.333,Z 581.552,A 0.000,B 0.000,C 90.000,E1 279.321} C_DIS
LIN {X 0.126,Y -461.508,Z 581.546,A 0.000,B 0.000,C 90.000,E1 278.276} C_DIS
LIN {X 0.230,Y -468.107,Z 581.540,A 0.000,B 0.000,C 90.000,E1 277.239} C_DIS
LIN {X 0.158,Y -472.643,Z 581.536,A 0.000,B 0.000,C 90.000,E1 276.486} C_DIS
LIN {X 0.065,Y -476.670,Z 581.532,A 0.000,B 0.000,C 90.000,E1 275.739} C_DIS
LIN {X 0.200,Y -479.010,Z 581.529,A 0.000,B 0.000,C 90.000,E1 275.220} C_DIS
LIN {X -0.129,Y -481.047,Z 581.526,A 0.000,B 0.000,C 90.000,E1 274.759} C_DIS
LIN {X -0.012,Y -482.773,Z 581.524,A 0.000,B 0.000,C 90.000,E1 274.245} C_DIS
LIN {X 0.154,Y -484.215,Z 581.521,A 0.000,B 0.000,C 90.000,E1 273.726} C_DIS
LIN {X -0.185,Y -485.394,Z 581.518,A 0.000,B 0.000,C 90.000,E1 273.269} C_DIS
LIN {X -0.004,Y -486.258,Z 581.515,A 0.000,B 0.000,C 90.000,E1 272.751} C_DIS
LIN {X 0.161,Y -486.788,Z 581.513,A 0.000,B 0.000,C 90.000,E1 272.236} C_DIS
LIN {X -0.137,Y -486.885,Z 581.510,A 0.000,B 0.000,C 90.000,E1 271.776} C_DIS
LIN {X 0.035,Y -486.508,Z 581.507,A 0.000,B 0.000,C 90.000,E1 271.260} C_DIS
LIN {X 0.211,Y -485.661,Z 581.504,A 0.000,B 0.000,C 90.000,E1 270.745} C_DIS
LIN {X -0.100,Y -484.224,Z 581.502,A 0.000,B 0.000,C 90.000,E1 270.286} C_DIS
LIN {X 0.069,Y -482.157,Z 581.499,A 0.000,B 0.000,C 90.000,E1 269.771} C_DIS
LIN {X 0.228,Y -479.451,Z 581.496,A 0.000,B 0.000,C 90.000,E1 269.255} C_DIS
LIN {X -0.111,Y -475.904,Z 581.493,A 0.000,B 0.000,C 90.000,E1 268.797} C_DIS
LIN {X 0.009,Y -471.332,Z 581.490,A 0.000,B 0.000,C 90.000,E1 268.282} C_DIS
LIN {X 0.118,Y -465.475,Z 581.488,A 0.000,B 0.000,C 90.000,E1 267.764} C_DIS
LIN {X 0.210,Y -462.453,Z 581.486,A 0.000,B 0.000,C 90.000,E1 267.535} C_DIS
LIN {X -0.158,Y -459.014,Z 581.485,A 0.000,B 0.000,C 90.000,E1 267.364} C_DIS
LIN {X 0.158,Y -452.144,Z 581.483,A 0.000,B 0.000,C 90.000,E1 266.963} C_DIS
LIN {X 0.094,Y -444.772,Z 581.482,A 0.000,B 0.000,C 90.000,E1 266.674} C_DIS
LIN {X 0.065,Y -437.113,Z 581.480,A 0.000,B 0.000,C 90.000,E1 266.445} C_DIS
LIN {X 0.022,Y -428.517,Z 581.479,A 0.000,B 0.000,C 90.000,E1 266.274} C_DIS
LIN {X -0.026,Y -419.216,Z 581.479,A 0.000,B 0.000,C 90.000,E1 266.159} C_DIS
LIN {X -0.060,Y -410.580,Z 581.478,A 0.000,B 0.000,C 90.000,E1 266.102} C_DIS
LIN {X -0.133,Y -406.454,Z 581.478,A 0.000,B 0.000,C 90.000,E1 266.102} C_DIS
LIN {X -0.092,Y -180.923,Z 581.478,A 0.000,B 0.000,C 90.000,E1 266.102} C_DIS
LIN {X -0.047,Y -180.873,Z 581.472,A 0.000,B 0.000,C 90.000,E1 265.065} C_DIS
LIN {X 0.036,Y -178.936,Z 581.443,A 0.000,B 0.000,C 90.000,E1 259.803} C_DIS
LIN {X -0.096,Y -175.985,Z 581.415,A 0.000,B 0.000,C 90.000,E1 254.755} C_DIS
LIN {X 0.018,Y -175.482,Z 581.410,A 0.000,B 0.000,C 90.000,E1 253.866} C_DIS
LIN {X 0.075,Y -172.228,Z 581.387,A 0.000,B 0.000,C 90.000,E1 249.571} C_DIS
LIN {X 0.052,Y -171.704,Z 581.382,A 0.000,B 0.000,C 90.000,E1 248.720} C_DIS
LIN {X -0.023,Y -167.299,Z 581.353,A 0.000,B 0.000,C 90.000,E1 243.563} C_DIS
LIN {X -0.016,Y -166.677,Z 581.348,A 0.000,B 0.000,C 90.000,E1 242.692} C_DIS
LIN {X -0.025,Y -162.659,Z 581.324,A 0.000,B 0.000,C 90.000,E1 238.329} C_DIS
LIN {X 0.037,Y -161.349,Z 581.314,A 0.000,B 0.000,C 90.000,E1 236.548} C_DIS
LIN {X 0.079,Y -157.343,Z 581.290,A 0.000,B 0.000,C 90.000,E1 232.110} C_DIS
LIN {X 0.011,Y -155.328,Z 581.275,A 0.000,B 0.000,C 90.000,E1 229.461} C_DIS
LIN {X -0.058,Y -151.680,Z 581.250,A 0.000,B 0.000,C 90.000,E1 225.000} C_DIS
LIN {X -0.010,Y -150.544,Z 581.240,A 0.000,B 0.000,C 90.000,E1 223.176} C_DIS
LIN {X 0.023,Y -147.270,Z 581.215,A 0.000,B 0.000,C 90.000,E1 218.624} C_DIS
LIN {X -0.004,Y -145.297,Z 581.194,A 0.000,B 0.000,C 90.000,E1 214.978} C_DIS
LIN {X -0.012,Y -142.392,Z 581.164,A 0.000,B 0.000,C 90.000,E1 209.461} C_DIS
LIN {X 0.034,Y -141.373,Z 581.148,A 0.000,B 0.000,C 90.000,E1 206.668} C_DIS
LIN {X 0.012,Y -139.346,Z 581.112,A 0.000,B 0.000,C 90.000,E1 200.174} C_DIS
LIN {X -0.046,Y -138.782,Z 581.097,A 0.000,B 0.000,C 90.000,E1 197.402} C_DIS
LIN {X 0.013,Y -138.343,Z 581.055,A 0.000,B 0.000,C 90.000,E1 189.905} C_DIS
LIN {X 0.033,Y -139.392,Z 581.008,A 0.000,B 0.000,C 90.000,E1 181.489} C_DIS
LIN {X -0.054,Y -141.291,Z 580.972,A 0.000,B 0.000,C 90.000,E1 175.008} C_DIS
LIN {X 0.045,Y -142.654,Z 580.957,A 0.000,B 0.000,C 90.000,E1 172.186} C_DIS
LIN {X -0.005,Y -144.993,Z 580.931,A 0.000,B 0.000,C 90.000,E1 167.589} C_DIS
LIN {X -0.016,Y -147.621,Z 580.911,A 0.000,B 0.000,C 90.000,E1 163.921} C_DIS
LIN {X 0.063,Y -150.247,Z 580.890,A 0.000,B 0.000,C 90.000,E1 160.242} C_DIS
LIN {X -0.064,Y -153.642,Z 580.870,A 0.000,B 0.000,C 90.000,E1 156.666} C_DIS
LIN {X -0.005,Y -157.057,Z 580.850,A 0.000,B 0.000,C 90.000,E1 153.050} C_DIS
LIN {X 0.074,Y -161.187,Z 580.830,A 0.000,B 0.000,C 90.000,E1 149.459} C_DIS
LIN {X 0.023,Y -163.280,Z 580.821,A 0.000,B 0.000,C 90.000,E1 147.709} C_DIS
LIN {X 0.033,Y -167.723,Z 580.801,A 0.000,B 0.000,C 90.000,E1 144.196} C_DIS
LIN {X -0.054,Y -171.542,Z 580.787,A 0.000,B 0.000,C 90.000,E1 141.618} C_DIS
LIN {X -0.012,Y -176.484,Z 580.768,A 0.000,B 0.000,C 90.000,E1 138.162} C_DIS
LIN {X -0.013,Y -180.781,Z 580.753,A 0.000,B 0.000,C 90.000,E1 135.607} C_DIS
LIN {X -0.026,Y -186.188,Z 580.735,A 0.000,B 0.000,C 90.000,E1 132.243} C_DIS
LIN {X -0.039,Y -191.396,Z 580.719,A 0.000,B 0.000,C 90.000,E1 129.402} C_DIS
LIN {X 0.019,Y -191.498,Z 580.719,A 0.000,B 0.000,C 90.000,E1 129.322} C_DIS
LIN {X -0.006,Y -288.917,Z 580.718,A 0.000,B 0.000,C 90.000,E1 129.322} C_DIS
LIN {X -0.025,Y -291.146,Z 580.718,A 0.000,B 0.000,C 90.000,E1 129.277} C_DIS
LIN {X -0.006,Y -296.904,Z 580.716,A 0.000,B 0.000,C 90.000,E1 128.910} C_DIS
LIN {X -0.093,Y -300.103,Z 580.714,A 0.000,B 0.000,C 90.000,E1 128.543} C_DIS
LIN {X 0.126,Y -302.049,Z 580.712,A 0.000,B 0.000,C 90.000,E1 128.177} C_DIS
LIN {X -0.081,Y -303.566,Z 580.710,A 0.000,B 0.000,C 90.000,E1 127.890} C_DIS
LIN {X 0.117,Y -304.779,Z 580.709,A 0.000,B 0.000,C 90.000,E1 127.523} C_DIS
LIN {X 0.027,Y -316.508,Z 580.687,A 0.000,B 0.000,C 90.000,E1 123.627} C_DIS
LIN {X 0.033,Y -326.695,Z 580.671,A 0.000,B 0.000,C 90.000,E1 120.747} C_DIS
LIN {X 0.180,Y -338.220,Z 580.655,A 0.000,B 0.000,C 90.000,E1 117.897} C_DIS
LIN {X 0.017,Y -351.191,Z 580.640,A 0.000,B 0.000,C 90.000,E1 115.155} C_DIS
LIN {X -0.140,Y -364.026,Z 580.626,A 0.000,B 0.000,C 90.000,E1 112.770} C_DIS
LIN {X 0.087,Y -378.187,Z 580.613,A 0.000,B 0.000,C 90.000,E1 110.375} C_DIS
LIN {X 0.192,Y -393.775,Z 580.600,A 0.000,B 0.000,C 90.000,E1 108.055} C_DIS
LIN {X -0.071,Y -410.906,Z 580.588,A 0.000,B 0.000,C 90.000,E1 105.843} C_DIS
LIN {X -0.034,Y -429.704,Z 580.576,A 0.000,B 0.000,C 90.000,E1 103.647} C_DIS
LIN {X -0.167,Y -449.738,Z 580.564,A 0.000,B 0.000,C 90.000,E1 101.591} C_DIS
LIN {X -0.008,Y -470.330,Z 580.554,A 0.000,B 0.000,C 90.000,E1 99.670} C_DIS
LIN {X 0.086,Y -475.245,Z 580.551,A 0.000,B 0.000,C 90.000,E1 99.208} C_DIS
LIN {X 0.030,Y -477.109,Z 580.550,A 0.000,B 0.000,C 90.000,E1 98.973} C_DIS
LIN {X -0.100,Y -478.524,Z 580.549,A 0.000,B 0.000,C 90.000,E1 98.746} C_DIS
LIN {X 0.113,Y -480.414,Z 580.546,A 0.000,B 0.000,C 90.000,E1 98.219} C_DIS
LIN {X -0.211,Y -481.193,Z 580.543,A 0.000,B 0.000,C 90.000,E1 97.757} C_DIS
LIN {X -0.047,Y -480.994,Z 580.540,A 0.000,B 0.000,C 90.000,E1 97.239} C_DIS
LIN {X 0.122,Y -479.788,Z 580.537,A 0.000,B 0.000,C 90.000,E1 96.720} C_DIS
LIN {X -0.005,Y -478.751,Z 580.536,A 0.000,B 0.000,C 90.000,E1 96.486} C_DIS
LIN {X -0.185,Y -477.355,Z 580.535,A 0.000,B 0.000,C 90.000,E1 96.258} C_DIS
LIN {X -0.135,Y -458.886,Z 580.521,A 0.000,B 0.000,C 90.000,E1 93.726} C_DIS
LIN {X -0.120,Y -449.027,Z 580.512,A 0.000,B 0.000,C 90.000,E1 92.178} C_DIS
LIN {X -0.184,Y -435.850,Z 580.499,A 0.000,B 0.000,C 90.000,E1 89.828} C_DIS
LIN {X 0.155,Y -428.237,Z 580.492,A 0.000,B 0.000,C 90.000,E1 88.453} C_DIS
LIN {X 0.092,Y -418.637,Z 580.483,A 0.000,B 0.000,C 90.000,E1 86.846} C_DIS
LIN {X 0.112,Y -404.490,Z 580.469,A 0.000,B 0.000,C 90.000,E1 84.375} C_DIS
LIN {X -0.156,Y -390.893,Z 580.455,A 0.000,B 0.000,C 90.000,E1 81.894} C_DIS
LIN {X 0.063,Y -379.094,Z 580.442,A 0.000,B 0.000,C 90.000,E1 79.577} C_DIS
LIN {X 0.199,Y -367.461,Z 580.429,A 0.000,B 0.000,C 90.000,E1 77.229} C_DIS
LIN {X 0.021,Y -351.128,Z 580.409,A 0.000,B 0.000,C 90.000,E1 73.685} C_DIS
LIN {X 0.098,Y -336.866,Z 580.389,A 0.000,B 0.000,C 90.000,E1 70.007} C_DIS
LIN {X -0.151,Y -324.395,Z 580.368,A 0.000,B 0.000,C 90.000,E1 66.305} C_DIS
LIN {X -0.162,Y -316.756,Z 580.354,A 0.000,B 0.000,C 90.000,E1 63.768} C_DIS
LIN {X -0.074,Y -309.325,Z 580.340,A 0.000,B 0.000,C 90.000,E1 61.179} C_DIS
LIN {X 0.121,Y -302.008,Z 580.325,A 0.000,B 0.000,C 90.000,E1 58.535} C_DIS
LIN {X -0.055,Y -293.205,Z 580.307,A 0.000,B 0.000,C 90.000,E1 55.261} C_DIS
LIN {X 0.048,Y -286.558,Z 580.292,A 0.000,B 0.000,C 90.000,E1 52.557} C_DIS
LIN {X 0.075,Y -281.546,Z 580.281,A 0.000,B 0.000,C 90.000,E1 50.517} C_DIS
LIN {X -0.047,Y -277.999,Z 580.273,A 0.000,B 0.000,C 90.000,E1 49.175} C_DIS
LIN {X -0.030,Y -274.249,Z 580.266,A 0.000,B 0.000,C 90.000,E1 47.796} C_DIS
LIN {X 0.125,Y -270.193,Z 580.258,A 0.000,B 0.000,C 90.000,E1 46.377} C_DIS
LIN {X -0.091,Y -264.662,Z 580.248,A 0.000,B 0.000,C 90.000,E1 44.676} C_DIS
LIN {X 0.013,Y -257.736,Z 580.236,A 0.000,B 0.000,C 90.000,E1 42.528} C_DIS
LIN {X 0.052,Y -247.516,Z 580.218,A 0.000,B 0.000,C 90.000,E1 39.277} C_DIS
LIN {X -0.082,Y -239.180,Z 580.202,A 0.000,B 0.000,C 90.000,E1 36.377} C_DIS
LIN {X 0.004,Y -229.739,Z 580.181,A 0.000,B 0.000,C 90.000,E1 32.625} C_DIS
LIN {X 0.003,Y -222.931,Z 580.164,A 0.000,B 0.000,C 90.000,E1 29.589} C_DIS
LIN {X 0.081,Y -216.896,Z 580.147,A 0.000,B 0.000,C 90.000,E1 26.488} C_DIS
LIN {X 0.060,Y -210.290,Z 580.126,A 0.000,B 0.000,C 90.000,E1 22.589} C_DIS
LIN {X -0.023,Y -206.072,Z 580.108,A 0.000,B 0.000,C 90.000,E1 19.450} C_DIS
LIN {X 0.091,Y -201.906,Z 580.086,A 0.000,B 0.000,C 90.000,E1 15.426} C_DIS
LIN {X 0.049,Y -198.204,Z 580.059,A 0.000,B 0.000,C 90.000,E1 10.602} C_DIS
LIN {X -0.047,Y -195.686,Z 580.023,A 0.000,B 0.000,C 90.000,E1 4.131} C_DIS
LIN {X 0.098,Y -197.240,Z 579.966,A 0.000,B 0.000,C 90.000,E1 353.799} C_DIS
LIN {X -0.078,Y -200.247,Z 579.939,A 0.000,B 0.000,C 90.000,E1 348.982} C_DIS
LIN {X -0.100,Y -204.570,Z 579.912,A 0.000,B 0.000,C 90.000,E1 344.157} C_DIS
LIN {X 0.016,Y -208.970,Z 579.890,A 0.000,B 0.000,C 90.000,E1 340.134} C_DIS
LIN {X 0.042,Y -214.214,Z 579.868,A 0.000,B 0.000,C 90.000,E1 336.177} C_DIS
LIN {X 0.005,Y -220.072,Z 579.846,A 0.000,B 0.000,C 90.000,E1 332.281} C_DIS
LIN {X 0.076,Y -226.551,Z 579.825,A 0.000,B 0.000,C 90.000,E1 328.408} C_DIS
LIN {X 0.058,Y -233.576,Z 579.803,A 0.000,B 0.000,C 90.000,E1 324.609} C_DIS
LIN {X -0.039,Y -240.986,Z 579.783,A 0.000,B 0.000,C 90.000,E1 320.884} C_DIS
LIN {X -0.016,Y -249.140,Z 579.762,A 0.000,B 0.000,C 90.000,E1 317.187} C_DIS
LIN {X 0.052,Y -258.250,Z 579.742,A 0.000,B 0.000,C 90.000,E1 313.542} C_DIS
LIN {X 0.056,Y -267.651,Z 579.724,A 0.000,B 0.000,C 90.000,E1 310.334} C_DIS
LIN {X -0.005,Y -278.600,Z 579.707,A 0.000,B 0.000,C 90.000,E1 307.202} C_DIS
LIN {X 0.019,Y -290.673,Z 579.690,A 0.000,B 0.000,C 90.000,E1 304.119} C_DIS
LIN {X -0.091,Y -304.007,Z 579.673,A 0.000,B 0.000,C 90.000,E1 301.131} C_DIS
LIN {X -0.012,Y -318.232,Z 579.657,A 0.000,B 0.000,C 90.000,E1 298.180} C_DIS
LIN {X -0.075,Y -331.714,Z 579.642,A 0.000,B 0.000,C 90.000,E1 295.643} C_DIS
LIN {X 0.066,Y -346.428,Z 579.629,A 0.000,B 0.000,C 90.000,E1 293.131} C_DIS
LIN {X -0.136,Y -362.712,Z 579.615,A 0.000,B 0.000,C 90.000,E1 290.737} C_DIS
LIN {X 0.069,Y -385.114,Z 579.599,A 0.000,B 0.000,C 90.000,E1 287.764} C_DIS
LIN {X -0.035,Y -399.247,Z 579.589,A 0.000,B 0.000,C 90.000,E1 286.079} C_DIS
LIN {X -0.106,Y -413.449,Z 579.580,A 0.000,B 0.000,C 90.000,E1 284.411} C_DIS
LIN {X -0.063,Y -427.489,Z 579.571,A 0.000,B 0.000,C 90.000,E1 282.771} C_DIS
LIN {X -0.191,Y -436.337,Z 579.565,A 0.000,B 0.000,C 90.000,E1 281.715} C_DIS
LIN {X -0.023,Y -446.731,Z 579.558,A 0.000,B 0.000,C 90.000,E1 280.366} C_DIS
LIN {X -0.032,Y -454.479,Z 579.552,A 0.000,B 0.000,C 90.000,E1 279.321} C_DIS
LIN {X 0.051,Y -461.643,Z 579.546,A 0.000,B 0.000,C 90.000,E1 278.276} C_DIS
LIN {X 0.154,Y -468.241,Z 579.540,A 0.000,B 0.000,C 90.000,E1 277.239} C_DIS
LIN {X 0.082,Y -472.752,Z 579.536,A 0.000,B 0.000,C 90.000,E1 276.486} C_DIS
LIN {X -0.010,Y -476.734,Z 579.532,A 0.000,B 0.000,C 90.000,E1 275.739} C_DIS
LIN {X 0.126,Y -479.084,Z 579.529,A 0.000,B 0.000,C 90.000,E1 275.220} C_DIS
LIN {X -0.204,Y -481.124,Z 579.526,A 0.000,B 0.000,C 90.000,E1 274.759} C_DIS
LIN {X -0.087,Y -482.860,Z 579.523,A 0.000,B 0.000,C 90.000,E1 274.245} C_DIS
LIN {X 0.079,Y -484.302,Z 579.521,A 0.000,B 0.000,C 90.000,E1 273.726} C_DIS
LIN {X 0.226,Y -485.474,Z 579.518,A 0.000,B 0.000,C 90.000,E1 273.212} C_DIS
LIN {X -0.077,Y -486.336,Z 579.515,A 0.000,B 0.000,C 90.000,E1 272.751} C_DIS
LIN {X 0.088,Y -486.858,Z 579.512,A 0.000,B 0.000,C 90.000,E1 272.236} C_DIS
LIN {X -0.210,Y -486.946,Z 579.510,A 0.000,B 0.000,C 90.000,E1 271.776} C_DIS
LIN {X -0.037,Y -486.560,Z 579.507,A 0.000,B 0.000,C 90.000,E1 271.260} C_DIS
LIN {X 0.140,Y -485.666,Z 579.504,A 0.000,B 0.000,C 90.000,E1 270.745} C_DIS
LIN {X -0.171,Y -484.191,Z 579.501,A 0.000,B 0.000,C 90.000,E1 270.286} C_DIS
LIN {X -0.001,Y -482.146,Z 579.499,A 0.000,B 0.000,C 90.000,E1 269.771} C_DIS
LIN {X 0.157,Y -479.351,Z 579.496,A 0.000,B 0.000,C 90.000,E1 269.255} C_DIS
LIN {X -0.181,Y -475.799,Z 579.493,A 0.000,B 0.000,C 90.000,E1 268.797} C_DIS
LIN {X 0.116,Y -473.612,Z 579.492,A 0.000,B 0.000,C 90.000,E1 268.511} C_DIS
LIN {X -0.208,Y -468.443,Z 579.489,A 0.000,B 0.000,C 90.000,E1 268.051} C_DIS
LIN {X 0.203,Y -462.377,Z 579.486,A 0.000,B 0.000,C 90.000,E1 267.535} C_DIS
LIN {X -0.212,Y -455.746,Z 579.484,A 0.000,B 0.000,C 90.000,E1 267.192} C_DIS
LIN {X 0.181,Y -452.172,Z 579.483,A 0.000,B 0.000,C 90.000,E1 266.963} C_DIS
LIN {X 0.109,Y -444.779,Z 579.482,A 0.000,B 0.000,C 90.000,E1 266.674} C_DIS
LIN {X 0.069,Y -437.114,Z 579.480,A 0.000,B 0.000,C 90.000,E1 266.445} C_DIS
LIN {X 0.024,Y -428.575,Z 579.479,A 0.000,B 0.000,C 90.000,E1 266.274} C_DIS
LIN {X -0.023,Y -419.338,Z 579.479,A 0.000,B 0.000,C 90.000,E1 266.159} C_DIS
LIN {X -0.065,Y -410.961,Z 579.478,A 0.000,B 0.000,C 90.000,E1 266.102} C_DIS
LIN {X -0.138,Y -406.858,Z 579.478,A 0.000,B 0.000,C 90.000,E1 266.102} C_DIS
LIN {X -0.094,Y -180.923,Z 579.478,A 0.000,B 0.000,C 90.000,E1 266.102} C_DIS
LIN {X -0.050,Y -180.873,Z 579.472,A 0.000,B 0.000,C 90.000,E1 265.065} C_DIS
LIN {X 0.033,Y -178.936,Z 579.443,A 0.000,B 0.000,C 90.000,E1 259.803} C_DIS
LIN {X -0.099,Y -175.985,Z 579.415,A 0.000,B 0.000,C 90.000,E1 254.755} C_DIS
LIN {X 0.016,Y -175.481,Z 579.410,A 0.000,B 0.000,C 90.000,E1 253.866} C_DIS
LIN {X 0.072,Y -172.227,Z 579.387,A 0.000,B 0.000,C 90.000,E1 249.571} C_DIS
LIN {X 0.049,Y -171.703,Z 579.382,A 0.000,B 0.000,C 90.000,E1 248.720} C_DIS
LIN {X -0.025,Y -167.298,Z 579.353,A 0.000,B 0.000,C 90.000,E1 243.563} C_DIS
LIN {X -0.019,Y -166.677,Z 579.348,A 0.000,B 0.000,C 90.000,E1 242.692} C_DIS
LIN {X -0.028,Y -162.659,Z 579.324,A 0.000,B 0.000,C 90.000,E1 238.329} C_DIS
LIN {X 0.035,Y -161.348,Z 579.314,A 0.000,B 0.000,C 90.000,E1 236.548} C_DIS
LIN {X 0.077,Y -157.342,Z 579.290,A 0.000,B 0.000,C 90.000,E1 232.110} C_DIS
LIN {X 0.009,Y -155.328,Z 579.275,A 0.000,B 0.000,C 90.000,E1 229.461} C_DIS
LIN {X -0.060,Y -151.679,Z 579.250,A 0.000,B 0.000,C 90.000,E1 225.000} C_DIS
LIN {X -0.012,Y -150.543,Z 579.240,A 0.000,B 0.000,C 90.000,E1 223.176} C_DIS
LIN {X 0.021,Y -147.270,Z 579.215,A 0.000,B 0.000,C 90.000,E1 218.624} C_DIS
LIN {X -0.007,Y -145.296,Z 579.194,A 0.000,B 0.000,C 90.000,E1 214.978} C_DIS
LIN {X -0.014,Y -142.392,Z 579.164,A 0.000,B 0.000,C 90.000,E1 209.461} C_DIS
LIN {X 0.032,Y -141.373,Z 579.148,A 0.000,B 0.000,C 90.000,E1 206.668} C_DIS
LIN {X 0.010,Y -139.346,Z 579.112,A 0.000,B 0.000,C 90.000,E1 200.174} C_DIS
LIN {X 0.015,Y -139.019,Z 579.102,A 0.000,B 0.000,C 90.000,E1 198.308} C_DIS
LIN {X 0.011,Y -138.343,Z 579.055,A 0.000,B 0.000,C 90.000,E1 189.905} C_DIS
LIN {X 0.030,Y -139.392,Z 579.008,A 0.000,B 0.000,C 90.000,E1 181.489} C_DIS
LIN {X -0.056,Y -141.291,Z 578.972,A 0.000,B 0.000,C 90.000,E1 175.008} C_DIS
LIN {X 0.043,Y -142.654,Z 578.957,A 0.000,B 0.000,C 90.000,E1 172.186} C_DIS
LIN {X -0.007,Y -144.994,Z 578.931,A 0.000,B 0.000,C 90.000,E1 167.589} C_DIS
LIN {X -0.018,Y -147.621,Z 578.911,A 0.000,B 0.000,C 90.000,E1 163.921} C_DIS
LIN {X 0.060,Y -150.248,Z 578.890,A 0.000,B 0.000,C 90.000,E1 160.242} C_DIS
LIN {X -0.066,Y -153.642,Z 578.870,A 0.000,B 0.000,C 90.000,E1 156.666} C_DIS
LIN {X -0.008,Y -157.058,Z 578.850,A 0.000,B 0.000,C 90.000,E1 153.050} C_DIS
LIN {X 0.072,Y -161.188,Z 578.830,A 0.000,B 0.000,C 90.000,E1 149.459} C_DIS
LIN {X 0.020,Y -163.281,Z 578.821,A 0.000,B 0.000,C 90.000,E1 147.709} C_DIS
LIN {X 0.030,Y -167.725,Z 578.801,A 0.000,B 0.000,C 90.000,E1 144.196} C_DIS
LIN {X -0.057,Y -171.543,Z 578.787,A 0.000,B 0.000,C 90.000,E1 141.618} C_DIS
LIN {X -0.015,Y -176.485,Z 578.768,A 0.000,B 0.000,C 90.000,E1 138.162} C_DIS
LIN {X -0.016,Y -180.783,Z 578.753,A 0.000,B 0.000,C 90.000,E1 135.607} C_DIS
LIN {X -0.028,Y -186.189,Z 578.735,A 0.000,B 0.000,C 90.000,E1 132.243} C_DIS
LIN {X -0.043,Y -191.397,Z 578.719,A 0.000,B 0.000,C 90.000,E1 129.402} C_DIS
LIN {X -0.008,Y -191.511,Z 578.718,A 0.000,B 0.000,C 90.000,E1 129.322} C_DIS
LIN {X -0.046,Y -288.266,Z 578.718,A 0.000,B 0.000,C 90.000,E1 129.322} C_DIS
LIN {X -0.030,Y -290.777,Z 578.718,A 0.000,B 0.000,C 90.000,E1 129.277} C_DIS
LIN {X -0.135,Y -294.557,Z 578.717,A 0.000,B 0.000,C 90.000,E1 129.116} C_DIS
LIN {X -0.010,Y -296.792,Z 578.716,A 0.000,B 0.000,C 90.000,E1 128.910} C_DIS
LIN {X -0.173,Y -300.664,Z 578.714,A 0.000,B 0.000,C 90.000,E1 128.463} C_DIS
LIN {X 0.007,Y -302.520,Z 578.712,A 0.000,B 0.000,C 90.000,E1 128.096} C_DIS
LIN {X 0.190,Y -303.969,Z 578.710,A 0.000,B 0.000,C 90.000,E1 127.729} C_DIS
LIN {X 0.161,Y -306.018,Z 578.706,A 0.000,B 0.000,C 90.000,E1 127.076} C_DIS
LIN {X 0.073,Y -315.784,Z 578.688,A 0.000,B 0.000,C 90.000,E1 123.833} C_DIS
LIN {X -0.217,Y -325.873,Z 578.672,A 0.000,B 0.000,C 90.000,E1 121.003} C_DIS
LIN {X -0.109,Y -337.298,Z 578.656,A 0.000,B 0.000,C 90.000,E1 118.153} C_DIS
LIN {X 0.160,Y -350.155,Z 578.641,A 0.000,B 0.000,C 90.000,E1 115.335} C_DIS
LIN {X -0.023,Y -362.883,Z 578.628,A 0.000,B 0.000,C 90.000,E1 112.950} C_DIS
LIN {X -0.177,Y -376.929,Z 578.614,A 0.000,B 0.000,C 90.000,E1 110.610} C_DIS
LIN {X -0.121,Y -392.394,Z 578.602,A 0.000,B 0.000,C 90.000,E1 108.290} C_DIS
LIN {X -0.042,Y -409.390,Z 578.589,A 0.000,B 0.000,C 90.000,E1 106.024} C_DIS
LIN {X -0.038,Y -428.044,Z 578.577,A 0.000,B 0.000,C 90.000,E1 103.828} C_DIS
LIN {X 0.168,Y -448.009,Z 578.565,A 0.000,B 0.000,C 90.000,E1 101.715} C_DIS
LIN {X -0.223,Y -468.558,Z 578.555,A 0.000,B 0.000,C 90.000,E1 99.849} C_DIS
LIN {X -0.081,Y -473.761,Z 578.552,A 0.000,B 0.000,C 90.000,E1 99.378} C_DIS
LIN {X -0.066,Y -475.893,Z 578.551,A 0.000,B 0.000,C 90.000,E1 99.151} C_DIS
LIN {X -0.203,Y -477.689,Z 578.549,A 0.000,B 0.000,C 90.000,E1 98.916} C_DIS
LIN {X 0.130,Y -479.037,Z 578.548,A 0.000,B 0.000,C 90.000,E1 98.624} C_DIS
LIN {X -0.199,Y -480.727,Z 578.545,A 0.000,B 0.000,C 90.000,E1 98.163} C_DIS
LIN {X -0.044,Y -481.341,Z 578.542,A 0.000,B 0.000,C 90.000,E1 97.644} C_DIS
LIN {X 0.123,Y -480.984,Z 578.540,A 0.000,B 0.000,C 90.000,E1 97.125} C_DIS
LIN {X -0.183,Y -479.600,Z 578.537,A 0.000,B 0.000,C 90.000,E1 96.663} C_DIS
LIN {X 0.166,Y -478.453,Z 578.536,A 0.000,B 0.000,C 90.000,E1 96.372} C_DIS
LIN {X -0.014,Y -476.921,Z 578.534,A 0.000,B 0.000,C 90.000,E1 96.144} C_DIS
LIN {X 0.235,Y -460.149,Z 578.521,A 0.000,B 0.000,C 90.000,E1 93.841} C_DIS
LIN {X 0.049,Y -451.710,Z 578.514,A 0.000,B 0.000,C 90.000,E1 92.579} C_DIS
LIN {X 0.125,Y -441.224,Z 578.504,A 0.000,B 0.000,C 90.000,E1 90.745} C_DIS
LIN {X 0.111,Y -433.897,Z 578.497,A 0.000,B 0.000,C 90.000,E1 89.427} C_DIS
LIN {X -0.004,Y -426.149,Z 578.490,A 0.000,B 0.000,C 90.000,E1 88.108} C_DIS
LIN {X 0.106,Y -413.351,Z 578.477,A 0.000,B 0.000,C 90.000,E1 85.927} C_DIS
LIN {X 0.029,Y -399.410,Z 578.464,A 0.000,B 0.000,C 90.000,E1 83.451} C_DIS
LIN {X 0.022,Y -387.438,Z 578.451,A 0.000,B 0.000,C 90.000,E1 81.197} C_DIS
LIN {X -0.147,Y -375.647,Z 578.438,A 0.000,B 0.000,C 90.000,E1 78.926} C_DIS
LIN {X -0.122,Y -361.288,Z 578.422,A 0.000,B 0.000,C 90.000,E1 75.992} C_DIS
LIN {X 0.078,Y -348.125,Z 578.405,A 0.000,B 0.000,C 90.000,E1 72.960} C_DIS
LIN {X 0.165,Y -334.276,Z 578.385,A 0.000,B 0.000,C 90.000,E1 69.263} C_DIS
LIN {X -0.027,Y -322.137,Z 578.364,A 0.000,B 0.000,C 90.000,E1 65.537} C_DIS
LIN {X -0.091,Y -314.590,Z 578.350,A 0.000,B 0.000,C 90.000,E1 62.999} C_DIS
LIN {X 0.088,Y -307.203,Z 578.336,A 0.000,B 0.000,C 90.000,E1 60.383} C_DIS
LIN {X -0.030,Y -299.913,Z 578.321,A 0.000,B 0.000,C 90.000,E1 57.788} C_DIS
LIN {X -0.101,Y -291.258,Z 578.303,A 0.000,B 0.000,C 90.000,E1 54.482} C_DIS
LIN {X -0.048,Y -284.615,Z 578.288,A 0.000,B 0.000,C 90.000,E1 51.778} C_DIS
LIN {X -0.097,Y -279.471,Z 578.276,A 0.000,B 0.000,C 90.000,E1 49.747} C_DIS
LIN {X 0.150,Y -275.814,Z 578.269,A 0.000,B 0.000,C 90.000,E1 48.324} C_DIS
LIN {X -0.061,Y -271.876,Z 578.261,A 0.000,B 0.000,C 90.000,E1 46.986} C_DIS
LIN {X -0.053,Y -266.495,Z 578.251,A 0.000,B 0.000,C 90.000,E1 45.243} C_DIS
LIN {X 0.091,Y -259.582,Z 578.240,A 0.000,B 0.000,C 90.000,E1 43.095} C_DIS
LIN {X -0.007,Y -249.264,Z 578.222,A 0.000,B 0.000,C 90.000,E1 39.886} C_DIS
LIN {X 0.047,Y -240.768,Z 578.205,A 0.000,B 0.000,C 90.000,E1 36.950} C_DIS
LIN {X -0.001,Y -233.013,Z 578.189,A 0.000,B 0.000,C 90.000,E1 33.992} C_DIS
LIN {X -0.111,Y -225.876,Z 578.172,A 0.000,B 0.000,C 90.000,E1 31.003} C_DIS
LIN {X 0.064,Y -219.469,Z 578.155,A 0.000,B 0.000,C 90.000,E1 27.897} C_DIS
LIN {X 0.015,Y -212.482,Z 578.133,A 0.000,B 0.000,C 90.000,E1 24.027} C_DIS
LIN {X 0.066,Y -207.719,Z 578.116,A 0.000,B 0.000,C 90.000,E1 20.865} C_DIS
LIN {X -0.030,Y -203.243,Z 578.094,A 0.000,B 0.000,C 90.000,E1 16.913} C_DIS
LIN {X 0.069,Y -199.129,Z 578.067,A 0.000,B 0.000,C 90.000,E1 12.063} C_DIS
LIN {X -0.074,Y -196.217,Z 578.036,A 0.000,B 0.000,C 90.000,E1 6.429} C_DIS
LIN {X 0.097,Y -197.233,Z 577.966,A 0.000,B 0.000,C 90.000,E1 353.799} C_DIS
LIN {X -0.079,Y -200.248,Z 577.939,A 0.000,B 0.000,C 90.000,E1 348.982} C_DIS
LIN {X -0.102,Y -204.572,Z 577.912,A 0.000,B 0.000,C 90.000,E1 344.157} C_DIS
LIN {X 0.015,Y -208.990,Z 577.890,A 0.000,B 0.000,C 90.000,E1 340.134} C_DIS
LIN {X 0.041,Y -214.222,Z 577.868,A 0.000,B 0.000,C 90.000,E1 336.177} C_DIS
LIN {X 0.005,Y -220.065,Z 577.846,A 0.000,B 0.000,C 90.000,E1 332.281} C_DIS
LIN {X 0.075,Y -226.548,Z 577.825,A 0.000,B 0.000,C 90.000,E1 328.408} C_DIS
LIN {X 0.057,Y -233.558,Z 577.803,A 0.000,B 0.000,C 90.000,E1 324.609} C_DIS
LIN {X -0.040,Y -240.963,Z 577.783,A 0.000,B 0.000,C 90.000,E1 320.884} C_DIS
LIN {X -0.017,Y -249.109,Z 577.762,A 0.000,B 0.000,C 90.000,E1 317.187} C_DIS
LIN {X 0.049,Y -258.208,Z 577.742,A 0.000,B 0.000,C 90.000,E1 313.542} C_DIS
LIN {X 0.052,Y -267.644,Z 577.724,A 0.000,B 0.000,C 90.000,E1 310.334} C_DIS
LIN {X -0.010,Y -278.581,Z 577.707,A 0.000,B 0.000,C 90.000,E1 307.202} C_DIS
LIN {X 0.013,Y -290.641,Z 577.690,A 0.000,B 0.000,C 90.000,E1 304.119} C_DIS
LIN {X -0.112,Y -302.427,Z 577.675,A 0.000,B 0.000,C 90.000,E1 301.465} C_DIS
LIN {X -0.021,Y -318.139,Z 577.657,A 0.000,B 0.000,C 90.000,E1 298.180} C_DIS
LIN {X -0.086,Y -331.620,Z 577.642,A 0.000,B 0.000,C 90.000,E1 295.643} C_DIS
LIN {X 0.051,Y -346.345,Z 577.629,A 0.000,B 0.000,C 90.000,E1 293.131} C_DIS
LIN {X -0.154,Y -362.660,Z 577.615,A 0.000,B 0.000,C 90.000,E1 290.737} C_DIS
LIN {X 0.050,Y -385.105,Z 577.599,A 0.000,B 0.000,C 90.000,E1 287.764} C_DIS
LIN {X -0.152,Y -399.362,Z 577.589,A 0.000,B 0.000,C 90.000,E1 286.079} C_DIS
LIN {X -0.117,Y -415.956,Z 577.578,A 0.000,B 0.000,C 90.000,E1 284.120} C_DIS
LIN {X -0.068,Y -427.517,Z 577.571,A 0.000,B 0.000,C 90.000,E1 282.771} C_DIS
LIN {X -0.216,Y -436.402,Z 577.565,A 0.000,B 0.000,C 90.000,E1 281.715} C_DIS
LIN {X 0.171,Y -444.792,Z 577.559,A 0.000,B 0.000,C 90.000,E1 280.602} C_DIS
LIN {X 0.145,Y -452.702,Z 577.553,A 0.000,B 0.000,C 90.000,E1 279.557} C_DIS
LIN {X 0.212,Y -459.998,Z 577.547,A 0.000,B 0.000,C 90.000,E1 278.511} C_DIS
LIN {X -0.162,Y -466.753,Z 577.542,A 0.000,B 0.000,C 90.000,E1 277.530} C_DIS
LIN {X 0.061,Y -472.830,Z 577.536,A 0.000,B 0.000,C 90.000,E1 276.486} C_DIS
LIN {X -0.030,Y -476.830,Z 577.532,A 0.000,B 0.000,C 90.000,E1 275.739} C_DIS
LIN {X 0.106,Y -479.145,Z 577.529,A 0.000,B 0.000,C 90.000,E1 275.220} C_DIS
LIN {X 0.255,Y -481.171,Z 577.526,A 0.000,B 0.000,C 90.000,E1 274.702} C_DIS
LIN {X -0.107,Y -482.925,Z 577.523,A 0.000,B 0.000,C 90.000,E1 274.245} C_DIS
LIN {X 0.060,Y -484.387,Z 577.521,A 0.000,B 0.000,C 90.000,E1 273.726} C_DIS
LIN {X 0.207,Y -485.553,Z 577.518,A 0.000,B 0.000,C 90.000,E1 273.212} C_DIS
LIN {X -0.095,Y -486.410,Z 577.515,A 0.000,B 0.000,C 90.000,E1 272.751} C_DIS
LIN {X 0.070,Y -486.918,Z 577.512,A 0.000,B 0.000,C 90.000,E1 272.236} C_DIS
LIN {X -0.228,Y -486.985,Z 577.510,A 0.000,B 0.000,C 90.000,E1 271.776} C_DIS
LIN {X -0.054,Y -486.579,Z 577.507,A 0.000,B 0.000,C 90.000,E1 271.260} C_DIS
LIN {X 0.122,Y -485.681,Z 577.504,A 0.000,B 0.000,C 90.000,E1 270.745} C_DIS
LIN {X -0.188,Y -484.176,Z 577.501,A 0.000,B 0.000,C 90.000,E1 270.286} C_DIS
LIN {X -0.018,Y -482.130,Z 577.499,A 0.000,B 0.000,C 90.000,E1 269.771} C_DIS
LIN {X 0.141,Y -479.312,Z 577.496,A 0.000,B 0.000,C 90.000,E1 269.255} C_DIS
LIN {X -0.198,Y -475.718,Z 577.493,A 0.000,B 0.000,C 90.000,E1 268.797} C_DIS
LIN {X 0.098,Y -473.551,Z 577.492,A 0.000,B 0.000,C 90.000,E1 268.511} C_DIS
LIN {X -0.211,Y -468.352,Z 577.489,A 0.000,B 0.000,C 90.000,E1 268.051} C_DIS
LIN {X 0.108,Y -465.324,Z 577.488,A 0.000,B 0.000,C 90.000,E1 267.764} C_DIS
LIN {X 0.201,Y -462.312,Z 577.486,A 0.000,B 0.000,C 90.000,E1 267.535} C_DIS
LIN {X 0.222,Y -455.705,Z 577.484,A 0.000,B 0.000,C 90.000,E1 267.135} C_DIS
LIN {X -0.080,Y -448.620,Z 577.482,A 0.000,B 0.000,C 90.000,E1 266.846} C_DIS
LIN {X 0.091,Y -441.245,Z 577.481,A 0.000,B 0.000,C 90.000,E1 266.560} C_DIS
LIN {X -0.161,Y -433.375,Z 577.480,A 0.000,B 0.000,C 90.000,E1 266.388} C_DIS
LIN {X 0.012,Y -424.867,Z 577.479,A 0.000,B 0.000,C 90.000,E1 266.216} C_DIS
LIN {X 0.090,Y -414.743,Z 577.478,A 0.000,B 0.000,C 90.000,E1 266.102} C_DIS
LIN {X -0.141,Y -407.500,Z 577.478,A 0.000,B 0.000,C 90.000,E1 266.102} C_DIS
LIN {X 0.084,Y -180.923,Z 577.478,A 0.000,B 0.000,C 90.000,E1 266.045} C_DIS
LIN {X -0.053,Y -180.872,Z 577.472,A 0.000,B 0.000,C 90.000,E1 265.065} C_DIS
LIN {X 0.030,Y -178.935,Z 577.443,A 0.000,B 0.000,C 90.000,E1 259.803} C_DIS
LIN {X 0.068,Y -175.984,Z 577.415,A 0.000,B 0.000,C 90.000,E1 254.700} C_DIS
LIN {X 0.012,Y -175.480,Z 577.410,A 0.000,B 0.000,C 90.000,E1 253.866} C_DIS
LIN {X 0.069,Y -172.227,Z 577.387,A 0.000,B 0.000,C 90.000,E1 249.571} C_DIS
LIN {X 0.046,Y -171.703,Z 577.382,A 0.000,B 0.000,C 90.000,E1 248.720} C_DIS
LIN {X -0.028,Y -167.298,Z 577.353,A 0.000,B 0.000,C 90.000,E1 243.563} C_DIS
LIN {X 0.054,Y -166.676,Z 577.348,A 0.000,B 0.000,C 90.000,E1 242.666} C_DIS
LIN {X -0.031,Y -162.658,Z 577.324,A 0.000,B 0.000,C 90.000,E1 238.329} C_DIS
LIN {X 0.032,Y -161.347,Z 577.314,A 0.000,B 0.000,C 90.000,E1 236.548} C_DIS
LIN {X 0.074,Y -157.342,Z 577.290,A 0.000,B 0.000,C 90.000,E1 232.110} C_DIS
LIN {X 0.006,Y -155.327,Z 577.275,A 0.000,B 0.000,C 90.000,E1 229.461} C_DIS
LIN {X -0.064,Y -151.679,Z 577.250,A 0.000,B 0.000,C 90.000,E1 225.000} C_DIS
LIN {X -0.016,Y -150.543,Z 577.240,A 0.000,B 0.000,C 90.000,E1 223.176} C_DIS
LIN {X 0.018,Y -147.269,Z 577.215,A 0.000,B 0.000,C 90.000,E1 218.624} C_DIS
LIN {X -0.009,Y -145.296,Z 577.194,A 0.000,B 0.000,C 90.000,E1 214.978} C_DIS
LIN {X -0.017,Y -142.392,Z 577.164,A 0.000,B 0.000,C 90.000,E1 209.461} C_DIS
LIN {X 0.029,Y -141.371,Z 577.148,A 0.000,B 0.000,C 90.000,E1 206.668} C_DIS
LIN {X 0.007,Y -139.346,Z 577.112,A 0.000,B 0.000,C 90.000,E1 200.174} C_DIS
LIN {X 0.012,Y -139.018,Z 577.102,A 0.000,B 0.000,C 90.000,E1 198.308} C_DIS
LIN {X 0.008,Y -138.342,Z 577.055,A 0.000,B 0.000,C 90.000,E1 189.905} C_DIS
LIN {X 0.028,Y -139.392,Z 577.008,A 0.000,B 0.000,C 90.000,E1 181.489} C_DIS
LIN {X -0.059,Y -141.292,Z 576.972,A 0.000,B 0.000,C 90.000,E1 175.008} C_DIS
LIN {X 0.040,Y -142.654,Z 576.957,A 0.000,B 0.000,C 90.000,E1 172.186} C_DIS
LIN {X -0.010,Y -144.994,Z 576.931,A 0.000,B 0.000,C 90.000,E1 167.589} C_DIS
LIN {X -0.021,Y -147.622,Z 576.911,A 0.000,B 0.000,C 90.000,E1 163.921} C_DIS
LIN {X 0.057,Y -150.249,Z 576.890,A 0.000,B 0.000,C 90.000,E1 160.242} C_DIS
LIN {X 0.072,Y -153.644,Z 576.870,A 0.000,B 0.000,C 90.000,E1 156.613} C_DIS
LIN {X -0.011,Y -157.060,Z 576.850,A 0.000,B 0.000,C 90.000,E1 153.050} C_DIS
LIN {X 0.069,Y -161.189,Z 576.830,A 0.000,B 0.000,C 90.000,E1 149.459} C_DIS
LIN {X 0.017,Y -163.282,Z 576.821,A 0.000,B 0.000,C 90.000,E1 147.709} C_DIS
LIN {X 0.027,Y -167.726,Z 576.801,A 0.000,B 0.000,C 90.000,E1 144.196} C_DIS
LIN {X -0.060,Y -171.544,Z 576.787,A 0.000,B 0.000,C 90.000,E1 141.618} C_DIS
LIN {X -0.018,Y -176.486,Z 576.768,A 0.000,B 0.000,C 90.000,E1 138.162} C_DIS
LIN {X 0.107,Y -180.784,Z 576.753,A 0.000,B 0.000,C 90.000,E1 135.567} C_DIS
LIN {X -0.032,Y -186.191,Z 576.735,A 0.000,B 0.000,C 90.000,E1 132.243} C_DIS
LIN {X -0.047,Y -191.398,Z 576.719,A 0.000,B 0.000,C 90.000,E1 129.402} C_DIS
LIN {X 0.090,Y -191.536,Z 576.718,A 0.000,B 0.000,C 90.000,E1 129.277} C_DIS
LIN {X 0.101,Y -288.886,Z 576.718,A 0.000,B 0.000,C 90.000,E1 129.277} C_DIS
LIN {X -0.037,Y -290.439,Z 576.718,A 0.000,B 0.000,C 90.000,E1 129.277} C_DIS
LIN {X -0.140,Y -294.425,Z 576.717,A 0.000,B 0.000,C 90.000,E1 129.116} C_DIS
LIN {X -0.015,Y -296.700,Z 576.716,A 0.000,B 0.000,C 90.000,E1 128.910} C_DIS
LIN {X -0.140,Y -300.565,Z 576.714,A 0.000,B 0.000,C 90.000,E1 128.463} C_DIS
LIN {X 0.057,Y -302.430,Z 576.712,A 0.000,B 0.000,C 90.000,E1 128.096} C_DIS
LIN {X -0.169,Y -303.887,Z 576.710,A 0.000,B 0.000,C 90.000,E1 127.810} C_DIS
LIN {X 0.043,Y -305.962,Z 576.706,A 0.000,B 0.000,C 90.000,E1 127.111} C_DIS
LIN {X -0.035,Y -315.723,Z 576.688,A 0.000,B 0.000,C 90.000,E1 123.865} C_DIS
LIN {X -0.149,Y -325.806,Z 576.672,A 0.000,B 0.000,C 90.000,E1 121.003} C_DIS
LIN {X -0.041,Y -337.226,Z 576.656,A 0.000,B 0.000,C 90.000,E1 118.153} C_DIS
LIN {X -0.088,Y -350.075,Z 576.641,A 0.000,B 0.000,C 90.000,E1 115.387} C_DIS
LIN {X 0.047,Y -362.798,Z 576.628,A 0.000,B 0.000,C 90.000,E1 112.950} C_DIS
LIN {X -0.107,Y -376.837,Z 576.614,A 0.000,B 0.000,C 90.000,E1 110.610} C_DIS
LIN {X -0.051,Y -392.295,Z 576.602,A 0.000,B 0.000,C 90.000,E1 108.290} C_DIS
LIN {X 0.029,Y -409.284,Z 576.589,A 0.000,B 0.000,C 90.000,E1 106.024} C_DIS
LIN {X 0.035,Y -427.930,Z 576.577,A 0.000,B 0.000,C 90.000,E1 103.828} C_DIS
LIN {X -0.203,Y -447.892,Z 576.565,A 0.000,B 0.000,C 90.000,E1 101.771} C_DIS
LIN {X -0.159,Y -468.438,Z 576.555,A 0.000,B 0.000,C 90.000,E1 99.849} C_DIS
LIN {X -0.017,Y -473.651,Z 576.552,A 0.000,B 0.000,C 90.000,E1 99.378} C_DIS
LIN {X -0.002,Y -475.840,Z 576.551,A 0.000,B 0.000,C 90.000,E1 99.151} C_DIS
LIN {X -0.124,Y -477.667,Z 576.549,A 0.000,B 0.000,C 90.000,E1 98.916} C_DIS
LIN {X 0.226,Y -479.040,Z 576.548,A 0.000,B 0.000,C 90.000,E1 98.624} C_DIS
LIN {X -0.103,Y -480.788,Z 576.545,A 0.000,B 0.000,C 90.000,E1 98.163} C_DIS
LIN {X 0.052,Y -481.450,Z 576.542,A 0.000,B 0.000,C 90.000,E1 97.644} C_DIS
LIN {X 0.220,Y -481.139,Z 576.540,A 0.000,B 0.000,C 90.000,E1 97.125} C_DIS
LIN {X -0.086,Y -479.807,Z 576.537,A 0.000,B 0.000,C 90.000,E1 96.663} C_DIS
LIN {X -0.211,Y -478.692,Z 576.536,A 0.000,B 0.000,C 90.000,E1 96.429} C_DIS
LIN {X 0.084,Y -477.201,Z 576.534,A 0.000,B 0.000,C 90.000,E1 96.144} C_DIS
LIN {X 0.121,Y -458.633,Z 576.520,A 0.000,B 0.000,C 90.000,E1 93.612} C_DIS
LIN {X 0.129,Y -448.776,Z 576.512,A 0.000,B 0.000,C 90.000,E1 92.064} C_DIS
LIN {X -0.115,Y -437.035,Z 576.500,A 0.000,B 0.000,C 90.000,E1 90.000} C_DIS
LIN {X -0.192,Y -429.472,Z 576.493,A 0.000,B 0.000,C 90.000,E1 88.682} C_DIS
LIN {X 0.173,Y -419.884,Z 576.484,A 0.000,B 0.000,C 90.000,E1 87.020} C_DIS
LIN {X -0.190,Y -405.694,Z 576.470,A 0.000,B 0.000,C 90.000,E1 84.609} C_DIS
LIN {X 0.019,Y -390.555,Z 576.454,A 0.000,B 0.000,C 90.000,E1 81.781} C_DIS
LIN {X -0.083,Y -378.708,Z 576.442,A 0.000,B 0.000,C 90.000,E1 79.511} C_DIS
LIN {X -0.022,Y -366.988,Z 576.429,A 0.000,B 0.000,C 90.000,E1 77.173} C_DIS
LIN {X -0.090,Y -353.241,Z 576.412,A 0.000,B 0.000,C 90.000,E1 74.212} C_DIS
LIN {X 0.049,Y -343.373,Z 576.399,A 0.000,B 0.000,C 90.000,E1 71.764} C_DIS
LIN {X -0.189,Y -332.220,Z 576.382,A 0.000,B 0.000,C 90.000,E1 68.720} C_DIS
LIN {X -0.030,Y -320.321,Z 576.361,A 0.000,B 0.000,C 90.000,E1 64.921} C_DIS
LIN {X -0.005,Y -312.831,Z 576.346,A 0.000,B 0.000,C 90.000,E1 62.359} C_DIS
LIN {X 0.123,Y -305.450,Z 576.332,A 0.000,B 0.000,C 90.000,E1 59.744} C_DIS
LIN {X -0.109,Y -296.437,Z 576.314,A 0.000,B 0.000,C 90.000,E1 56.501} C_DIS
LIN {X -0.092,Y -289.652,Z 576.299,A 0.000,B 0.000,C 90.000,E1 53.829} C_DIS
LIN {X 0.099,Y -283.008,Z 576.284,A 0.000,B 0.000,C 90.000,E1 51.090} C_DIS
LIN {X 0.024,Y -277.720,Z 576.273,A 0.000,B 0.000,C 90.000,E1 49.057} C_DIS
LIN {X 0.042,Y -273.906,Z 576.265,A 0.000,B 0.000,C 90.000,E1 47.676} C_DIS
LIN {X 0.011,Y -269.801,Z 576.257,A 0.000,B 0.000,C 90.000,E1 46.296} C_DIS
LIN {X -0.023,Y -264.231,Z 576.247,A 0.000,B 0.000,C 90.000,E1 44.555} C_DIS
LIN {X -0.068,Y -256.089,Z 576.234,A 0.000,B 0.000,C 90.000,E1 42.081} C_DIS
LIN {X -0.081,Y -247.079,Z 576.218,A 0.000,B 0.000,C 90.000,E1 39.197} C_DIS
LIN {X 0.111,Y -238.741,Z 576.201,A 0.000,B 0.000,C 90.000,E1 36.217} C_DIS
LIN {X 0.045,Y -229.323,Z 576.181,A 0.000,B 0.000,C 90.000,E1 32.498} C_DIS
LIN {X 0.034,Y -222.520,Z 576.164,A 0.000,B 0.000,C 90.000,E1 29.461} C_DIS
LIN {X 0.102,Y -216.514,Z 576.147,A 0.000,B 0.000,C 90.000,E1 26.360} C_DIS
LIN {X 0.068,Y -209.858,Z 576.125,A 0.000,B 0.000,C 90.000,E1 22.461} C_DIS
LIN {X -0.040,Y -206.653,Z 576.112,A 0.000,B 0.000,C 90.000,E1 20.120} C_DIS
LIN {X -0.042,Y -202.421,Z 576.090,A 0.000,B 0.000,C 90.000,E1 16.134} C_DIS
LIN {X -0.023,Y -198.551,Z 576.063,A 0.000,B 0.000,C 90.000,E1 11.299} C_DIS
LIN {X -0.084,Y -195.775,Z 576.027,A 0.000,B 0.000,C 90.000,E1 4.821} C_DIS
LIN {X 0.096,Y -197.228,Z 575.966,A 0.000,B 0.000,C 90.000,E1 353.799} C_DIS
LIN {X 0.117,Y -200.250,Z 575.939,A 0.000,B 0.000,C 90.000,E1 348.926} C_DIS
LIN {X -0.102,Y -204.574,Z 575.912,A 0.000,B 0.000,C 90.000,E1 344.157} C_DIS
LIN {X 0.015,Y -209.007,Z 575.890,A 0.000,B 0.000,C 90.000,E1 340.134} C_DIS
LIN {X 0.041,Y -214.227,Z 575.868,A 0.000,B 0.000,C 90.000,E1 336.177} C_DIS
LIN {X 0.005,Y -220.053,Z 575.846,A 0.000,B 0.000,C 90.000,E1 332.281} C_DIS
LIN {X 0.074,Y -226.537,Z 575.825,A 0.000,B 0.000,C 90.000,E1 328.408} C_DIS
LIN {X 0.056,Y -233.538,Z 575.803,A 0.000,B 0.000,C 90.000,E1 324.609} C_DIS
LIN {X -0.042,Y -240.947,Z 575.783,A 0.000,B 0.000,C 90.000,E1 320.884} C_DIS
LIN {X -0.020,Y -249.077,Z 575.762,A 0.000,B 0.000,C 90.000,E1 317.187} C_DIS
LIN {X 0.044,Y -258.178,Z 575.742,A 0.000,B 0.000,C 90.000,E1 313.542} C_DIS
LIN {X -0.017,Y -266.527,Z 575.726,A 0.000,B 0.000,C 90.000,E1 310.701} C_DIS
LIN {X -0.079,Y -274.787,Z 575.712,A 0.000,B 0.000,C 90.000,E1 308.257} C_DIS
LIN {X -0.098,Y -287.810,Z 575.693,A 0.000,B 0.000,C 90.000,E1 304.818} C_DIS
LIN {X -0.133,Y -300.891,Z 575.677,A 0.000,B 0.000,C 90.000,E1 301.799} C_DIS
LIN {X 0.056,Y -316.421,Z 575.658,A 0.000,B 0.000,C 90.000,E1 298.487} C_DIS
LIN {X 0.096,Y -329.742,Z 575.644,A 0.000,B 0.000,C 90.000,E1 295.924} C_DIS
LIN {X 0.035,Y -346.259,Z 575.629,A 0.000,B 0.000,C 90.000,E1 293.131} C_DIS
LIN {X -0.172,Y -362.610,Z 575.615,A 0.000,B 0.000,C 90.000,E1 290.737} C_DIS
LIN {X 0.030,Y -385.100,Z 575.599,A 0.000,B 0.000,C 90.000,E1 287.764} C_DIS
LIN {X -0.174,Y -399.355,Z 575.589,A 0.000,B 0.000,C 90.000,E1 286.079} C_DIS
LIN {X -0.140,Y -416.002,Z 575.578,A 0.000,B 0.000,C 90.000,E1 284.120} C_DIS
LIN {X 0.149,Y -427.749,Z 575.571,A 0.000,B 0.000,C 90.000,E1 282.715} C_DIS
LIN {X 0.011,Y -436.660,Z 575.565,A 0.000,B 0.000,C 90.000,E1 281.658} C_DIS
LIN {X 0.191,Y -447.101,Z 575.557,A 0.000,B 0.000,C 90.000,E1 280.310} C_DIS
LIN {X 0.191,Y -454.834,Z 575.552,A 0.000,B 0.000,C 90.000,E1 279.265} C_DIS
LIN {X -0.176,Y -461.997,Z 575.546,A 0.000,B 0.000,C 90.000,E1 278.276} C_DIS
LIN {X -0.071,Y -468.541,Z 575.540,A 0.000,B 0.000,C 90.000,E1 277.239} C_DIS
LIN {X -0.141,Y -473.022,Z 575.536,A 0.000,B 0.000,C 90.000,E1 276.486} C_DIS
LIN {X -0.232,Y -476.997,Z 575.532,A 0.000,B 0.000,C 90.000,E1 275.739} C_DIS
LIN {X -0.097,Y -479.298,Z 575.529,A 0.000,B 0.000,C 90.000,E1 275.220} C_DIS
LIN {X 0.053,Y -481.316,Z 575.526,A 0.000,B 0.000,C 90.000,E1 274.702} C_DIS
LIN {X 0.172,Y -483.059,Z 575.523,A 0.000,B 0.000,C 90.000,E1 274.188} C_DIS
LIN {X -0.142,Y -484.487,Z 575.521,A 0.000,B 0.000,C 90.000,E1 273.726} C_DIS
LIN {X 0.006,Y -485.655,Z 575.518,A 0.000,B 0.000,C 90.000,E1 273.212} C_DIS
LIN {X 0.188,Y -486.496,Z 575.515,A 0.000,B 0.000,C 90.000,E1 272.694} C_DIS
LIN {X -0.132,Y -486.950,Z 575.512,A 0.000,B 0.000,C 90.000,E1 272.236} C_DIS
LIN {X 0.057,Y -487.011,Z 575.510,A 0.000,B 0.000,C 90.000,E1 271.718} C_DIS
LIN {X 0.232,Y -486.578,Z 575.507,A 0.000,B 0.000,C 90.000,E1 271.203} C_DIS
LIN {X -0.078,Y -485.652,Z 575.504,A 0.000,B 0.000,C 90.000,E1 270.745} C_DIS
LIN {X 0.097,Y -484.119,Z 575.501,A 0.000,B 0.000,C 90.000,E1 270.229} C_DIS
LIN {X -0.217,Y -481.999,Z 575.499,A 0.000,B 0.000,C 90.000,E1 269.771} C_DIS
LIN {X -0.057,Y -479.165,Z 575.496,A 0.000,B 0.000,C 90.000,E1 269.255} C_DIS
LIN {X -0.227,Y -477.432,Z 575.494,A 0.000,B 0.000,C 90.000,E1 269.026} C_DIS
LIN {X -0.099,Y -473.249,Z 575.492,A 0.000,B 0.000,C 90.000,E1 268.511} C_DIS
LIN {X 0.195,Y -470.781,Z 575.490,A 0.000,B 0.000,C 90.000,E1 268.224} C_DIS
LIN {X -0.118,Y -464.948,Z 575.487,A 0.000,B 0.000,C 90.000,E1 267.764} C_DIS
LIN {X -0.015,Y -461.896,Z 575.486,A 0.000,B 0.000,C 90.000,E1 267.535} C_DIS
LIN {X 0.086,Y -458.441,Z 575.485,A 0.000,B 0.000,C 90.000,E1 267.306} C_DIS
LIN {X -0.030,Y -451.458,Z 575.483,A 0.000,B 0.000,C 90.000,E1 266.963} C_DIS
LIN {X -0.027,Y -444.237,Z 575.482,A 0.000,B 0.000,C 90.000,E1 266.674} C_DIS
LIN {X -0.042,Y -436.402,Z 575.480,A 0.000,B 0.000,C 90.000,E1 266.445} C_DIS
LIN {X -0.018,Y -428.440,Z 575.479,A 0.000,B 0.000,C 90.000,E1 266.274} C_DIS
LIN {X -0.082,Y -418.893,Z 575.479,A 0.000,B 0.000,C 90.000,E1 266.159} C_DIS
LIN {X -0.119,Y -409.191,Z 575.478,A 0.000,B 0.000,C 90.000,E1 266.102} C_DIS
LIN {X -0.191,Y -404.338,Z 575.478,A 0.000,B 0.000,C 90.000,E1 266.102} C_DIS
LIN {X 0.062,Y -180.923,Z 575.478,A 0.000,B 0.000,C 90.000,E1 266.045} C_DIS
LIN {X -0.074,Y -180.871,Z 575.472,A 0.000,B 0.000,C 90.000,E1 265.065} C_DIS
LIN {X 0.009,Y -178.933,Z 575.443,A 0.000,B 0.000,C 90.000,E1 259.803} C_DIS
LIN {X 0.047,Y -175.981,Z 575.415,A 0.000,B 0.000,C 90.000,E1 254.700} C_DIS
LIN {X -0.008,Y -175.475,Z 575.410,A 0.000,B 0.000,C 90.000,E1 253.866} C_DIS
LIN {X 0.049,Y -172.222,Z 575.387,A 0.000,B 0.000,C 90.000,E1 249.571} C_DIS
LIN {X 0.026,Y -171.698,Z 575.382,A 0.000,B 0.000,C 90.000,E1 248.720} C_DIS
LIN {X -0.048,Y -167.293,Z 575.353,A 0.000,B 0.000,C 90.000,E1 243.563} C_DIS
LIN {X 0.035,Y -166.670,Z 575.348,A 0.000,B 0.000,C 90.000,E1 242.666} C_DIS
LIN {X -0.050,Y -162.653,Z 575.324,A 0.000,B 0.000,C 90.000,E1 238.329} C_DIS
LIN {X 0.012,Y -161.341,Z 575.314,A 0.000,B 0.000,C 90.000,E1 236.548} C_DIS
LIN {X 0.055,Y -157.336,Z 575.290,A 0.000,B 0.000,C 90.000,E1 232.110} C_DIS
LIN {X -0.013,Y -155.320,Z 575.275,A 0.000,B 0.000,C 90.000,E1 229.461} C_DIS
LIN {X -0.081,Y -151.674,Z 575.250,A 0.000,B 0.000,C 90.000,E1 225.000} C_DIS
LIN {X -0.034,Y -150.538,Z 575.240,A 0.000,B 0.000,C 90.000,E1 223.176} C_DIS
LIN {X -0.001,Y -147.264,Z 575.215,A 0.000,B 0.000,C 90.000,E1 218.624} C_DIS
LIN {X -0.027,Y -145.291,Z 575.194,A 0.000,B 0.000,C 90.000,E1 214.978} C_DIS
LIN {X -0.036,Y -142.389,Z 575.164,A 0.000,B 0.000,C 90.000,E1 209.461} C_DIS
LIN {X 0.012,Y -141.368,Z 575.148,A 0.000,B 0.000,C 90.000,E1 206.668} C_DIS
LIN {X -0.011,Y -139.345,Z 575.112,A 0.000,B 0.000,C 90.000,E1 200.174} C_DIS
LIN {X -0.005,Y -139.016,Z 575.102,A 0.000,B 0.000,C 90.000,E1 198.308} C_DIS
LIN {X -0.009,Y -138.343,Z 575.055,A 0.000,B 0.000,C 90.000,E1 189.905} C_DIS
LIN {X 0.010,Y -139.394,Z 575.008,A 0.000,B 0.000,C 90.000,E1 181.489} C_DIS
LIN {X 0.064,Y -141.295,Z 574.972,A 0.000,B 0.000,C 90.000,E1 174.951} C_DIS
LIN {X 0.022,Y -142.657,Z 574.957,A 0.000,B 0.000,C 90.000,E1 172.186} C_DIS
LIN {X -0.029,Y -144.999,Z 574.931,A 0.000,B 0.000,C 90.000,E1 167.589} C_DIS
LIN {X -0.039,Y -147.626,Z 574.911,A 0.000,B 0.000,C 90.000,E1 163.921} C_DIS
LIN {X 0.039,Y -150.254,Z 574.890,A 0.000,B 0.000,C 90.000,E1 160.242} C_DIS
LIN {X 0.053,Y -153.652,Z 574.870,A 0.000,B 0.000,C 90.000,E1 156.613} C_DIS
LIN {X -0.030,Y -157.066,Z 574.850,A 0.000,B 0.000,C 90.000,E1 153.050} C_DIS
LIN {X 0.049,Y -161.198,Z 574.830,A 0.000,B 0.000,C 90.000,E1 149.459} C_DIS
LIN {X -0.003,Y -163.290,Z 574.821,A 0.000,B 0.000,C 90.000,E1 147.709} C_DIS
LIN {X 0.007,Y -167.735,Z 574.801,A 0.000,B 0.000,C 90.000,E1 144.196} C_DIS
LIN {X -0.080,Y -171.554,Z 574.787,A 0.000,B 0.000,C 90.000,E1 141.618} C_DIS
LIN {X -0.038,Y -176.497,Z 574.768,A 0.000,B 0.000,C 90.000,E1 138.162} C_DIS
LIN {X 0.086,Y -180.795,Z 574.753,A 0.000,B 0.000,C 90.000,E1 135.567} C_DIS
LIN {X -0.053,Y -186.203,Z 574.735,A 0.000,B 0.000,C 90.000,E1 132.243} C_DIS
LIN {X 0.079,Y -191.409,Z 574.719,A 0.000,B 0.000,C 90.000,E1 129.358} C_DIS
LIN {X 0.068,Y -191.546,Z 574.718,A 0.000,B 0.000,C 90.000,E1 129.277} C_DIS
LIN {X 0.068,Y -288.379,Z 574.718,A 0.000,B 0.000,C 90.000,E1 129.277} C_DIS
LIN {X -0.071,Y -290.288,Z 574.718,A 0.000,B 0.000,C 90.000,E1 129.277} C_DIS
LIN {X 0.055,Y -294.372,Z 574.717,A 0.000,B 0.000,C 90.000,E1 129.072} C_DIS
LIN {X -0.048,Y -296.664,Z 574.716,A 0.000,B 0.000,C 90.000,E1 128.910} C_DIS
LIN {X -0.158,Y -300.526,Z 574.714,A 0.000,B 0.000,C 90.000,E1 128.463} C_DIS
LIN {X 0.047,Y -302.395,Z 574.712,A 0.000,B 0.000,C 90.000,E1 128.096} C_DIS
LIN {X -0.173,Y -303.856,Z 574.710,A 0.000,B 0.000,C 90.000,E1 127.810} C_DIS
LIN {X 0.039,Y -305.944,Z 574.706,A 0.000,B 0.000,C 90.000,E1 127.111} C_DIS
LIN {X -0.040,Y -315.705,Z 574.688,A 0.000,B 0.000,C 90.000,E1 123.865} C_DIS
LIN {X -0.153,Y -325.788,Z 574.672,A 0.000,B 0.000,C 90.000,E1 121.003} C_DIS
LIN {X -0.047,Y -337.207,Z 574.656,A 0.000,B 0.000,C 90.000,E1 118.153} C_DIS
LIN {X 0.223,Y -350.058,Z 574.641,A 0.000,B 0.000,C 90.000,E1 115.335} C_DIS
LIN {X 0.039,Y -362.781,Z 574.628,A 0.000,B 0.000,C 90.000,E1 112.950} C_DIS
LIN {X -0.115,Y -376.820,Z 574.614,A 0.000,B 0.000,C 90.000,E1 110.610} C_DIS
LIN {X -0.059,Y -392.278,Z 574.602,A 0.000,B 0.000,C 90.000,E1 108.290} C_DIS
LIN {X 0.020,Y -409.268,Z 574.589,A 0.000,B 0.000,C 90.000,E1 106.024} C_DIS
LIN {X 0.024,Y -427.914,Z 574.577,A 0.000,B 0.000,C 90.000,E1 103.828} C_DIS
LIN {X -0.213,Y -447.877,Z 574.565,A 0.000,B 0.000,C 90.000,E1 101.771} C_DIS
LIN {X -0.170,Y -468.423,Z 574.555,A 0.000,B 0.000,C 90.000,E1 99.849} C_DIS
LIN {X -0.028,Y -473.639,Z 574.552,A 0.000,B 0.000,C 90.000,E1 99.378} C_DIS
LIN {X -0.014,Y -475.862,Z 574.551,A 0.000,B 0.000,C 90.000,E1 99.151} C_DIS
LIN {X -0.116,Y -477.698,Z 574.549,A 0.000,B 0.000,C 90.000,E1 98.916} C_DIS
LIN {X 0.252,Y -479.084,Z 574.548,A 0.000,B 0.000,C 90.000,E1 98.624} C_DIS
LIN {X -0.077,Y -480.870,Z 574.545,A 0.000,B 0.000,C 90.000,E1 98.163} C_DIS
LIN {X 0.079,Y -481.565,Z 574.543,A 0.000,B 0.000,C 90.000,E1 97.644} C_DIS
LIN {X -0.231,Y -481.284,Z 574.540,A 0.000,B 0.000,C 90.000,E1 97.182} C_DIS
LIN {X -0.059,Y -479.988,Z 574.537,A 0.000,B 0.000,C 90.000,E1 96.663} C_DIS
LIN {X -0.184,Y -478.895,Z 574.536,A 0.000,B 0.000,C 90.000,E1 96.429} C_DIS
